(* Logix 5000 project; controller reports 1756-L63 rev 20.11; software revision 20.04; part 4 of 52 *)

        [307].log_data[0].time := 900.0, [307].log_data[0].valid := 1, [307].log_data[1].valid := 1, [307].log_data[2].valid := 1, [307].log_data[3].valid := 1, [307].log_data[4].valid := 1, [307].log_data[5].valid := 1, [307].log_data[6].valid := 1, [307].log_data[7].valid := 1, [307].log_data[8].valid := 1, [307].log_data[9].valid := 1, [307].log_data[10].valid := 1, [307].log_data[11].valid := 1, [307].log_data[12].valid := 1, [307].log_data[13].valid := 1, [307].log_data[14].valid := 1, [307].log_data[15].valid := 1, [307].log_data[16].valid := 1, [307].log_data[17].valid := 1, [307].log_data[18].valid := 1, [307].log_data[19].valid := 1, [307].time.Year := 2023, [307].time.Month := 1, [307].time.Day := 19, [307].time.Hour := 5, [307].time.Minute := 14, [307].time.Second := 59, [308].log_data[0].min := 1.0, [308].log_data[0].max := 1.0, [308].log_data[0].total := 900.0, [308].log_data[0].time := 900.0, [308].log_data[0].minminute := 15, [308].log_data[0].maxminute := 15, [308].log_data[0].valid := 1, [308].log_data[1].valid := 1, [308].log_data[2].valid := 1, [308].log_data[3].valid := 1, [308].log_data[4].valid := 1, [308].log_data[5].valid := 1, [308].log_data[6].valid := 1, [308].log_data[7].valid := 1, [308].log_data[8].valid := 1, [308].log_data[9].valid := 1, [308].log_data[10].valid := 1, [308].log_data[11].valid := 1, [308].log_data[12].valid := 1, [308].log_data[13].valid := 1, [308].log_data[14].valid := 1, [308].log_data[15].valid := 1, [308].log_data[16].valid := 1, [308].log_data[17].valid := 1, [308].log_data[18].valid := 1, [308].log_data[19].valid := 1, [308].time.Year := 2023, [308].time.Month := 1, [308].time.Day := 19, [308].time.Hour := 5, [308].time.Minute := 29, [308].time.Second := 59, [309].log_data[0].min := 1.0,
        [309].log_data[0].max := 1.0, [309].log_data[0].total := 900.0, [309].log_data[0].time := 900.0, [309].log_data[0].minminute := 30, [309].log_data[0].maxminute := 30, [309].log_data[0].valid := 1, [309].log_data[1].valid := 1, [309].log_data[2].valid := 1, [309].log_data[3].valid := 1, [309].log_data[4].valid := 1, [309].log_data[5].valid := 1, [309].log_data[6].valid := 1, [309].log_data[7].valid := 1, [309].log_data[8].valid := 1, [309].log_data[9].valid := 1, [309].log_data[10].valid := 1, [309].log_data[11].valid := 1, [309].log_data[12].valid := 1, [309].log_data[13].valid := 1, [309].log_data[14].valid := 1, [309].log_data[15].valid := 1, [309].log_data[16].valid := 1, [309].log_data[17].valid := 1, [309].log_data[18].valid := 1, [309].log_data[19].valid := 1, [309].time.Year := 2023, [309].time.Month := 1, [309].time.Day := 19, [309].time.Hour := 5, [309].time.Minute := 44, [309].time.Second := 59, [310].log_data[0].min := 1.0, [310].log_data[0].max := 1.0, [310].log_data[0].total := 900.0, [310].log_data[0].time := 900.0, [310].log_data[0].minminute := 45, [310].log_data[0].maxminute := 45, [310].log_data[0].valid := 1, [310].log_data[1].valid := 1, [310].log_data[2].valid := 1, [310].log_data[3].valid := 1, [310].log_data[4].valid := 1, [310].log_data[5].valid := 1, [310].log_data[6].valid := 1, [310].log_data[7].valid := 1, [310].log_data[8].valid := 1, [310].log_data[9].valid := 1, [310].log_data[10].valid := 1, [310].log_data[11].valid := 1, [310].log_data[12].valid := 1, [310].log_data[13].valid := 1, [310].log_data[14].valid := 1, [310].log_data[15].valid := 1, [310].log_data[16].valid := 1, [310].log_data[17].valid := 1, [310].log_data[18].valid := 1, [310].log_data[19].valid := 1, [310].time.Year := 2023, [310].time.Month := 1, [310].time.Day := 19,
        [310].time.Hour := 5, [310].time.Minute := 59, [310].time.Second := 59, [311].log_data[0].min := 1.0, [311].log_data[0].max := 1.0, [311].log_data[0].total := 900.0, [311].log_data[0].time := 900.0, [311].log_data[0].valid := 1, [311].log_data[1].valid := 1, [311].log_data[2].valid := 1, [311].log_data[3].valid := 1, [311].log_data[4].valid := 1, [311].log_data[5].valid := 1, [311].log_data[6].valid := 1, [311].log_data[7].valid := 1, [311].log_data[8].valid := 1, [311].log_data[9].valid := 1, [311].log_data[10].valid := 1, [311].log_data[11].valid := 1, [311].log_data[12].valid := 1, [311].log_data[13].valid := 1, [311].log_data[14].valid := 1, [311].log_data[15].valid := 1, [311].log_data[16].valid := 1, [311].log_data[17].valid := 1, [311].log_data[18].valid := 1, [311].log_data[19].valid := 1, [311].time.Year := 2023, [311].time.Month := 1, [311].time.Day := 19, [311].time.Hour := 6, [311].time.Minute := 14, [311].time.Second := 59, [312].log_data[0].min := 1.0, [312].log_data[0].max := 1.0, [312].log_data[0].total := 900.0, [312].log_data[0].time := 900.0, [312].log_data[0].minminute := 15, [312].log_data[0].maxminute := 15, [312].log_data[0].valid := 1, [312].log_data[1].valid := 1, [312].log_data[2].valid := 1, [312].log_data[3].valid := 1, [312].log_data[4].valid := 1, [312].log_data[5].valid := 1, [312].log_data[6].valid := 1, [312].log_data[7].valid := 1, [312].log_data[8].valid := 1, [312].log_data[9].valid := 1, [312].log_data[10].valid := 1, [312].log_data[11].valid := 1, [312].log_data[12].valid := 1, [312].log_data[13].valid := 1, [312].log_data[14].valid := 1, [312].log_data[15].valid := 1, [312].log_data[16].valid := 1, [312].log_data[17].valid := 1, [312].log_data[18].valid := 1, [312].log_data[19].valid := 1, [312].time.Year := 2023,
        [312].time.Month := 1, [312].time.Day := 19, [312].time.Hour := 6, [312].time.Minute := 29, [312].time.Second := 59, [313].log_data[0].min := 1.0, [313].log_data[0].max := 1.0, [313].log_data[0].total := 900.0, [313].log_data[0].time := 900.0, [313].log_data[0].minminute := 30, [313].log_data[0].maxminute := 30, [313].log_data[0].valid := 1, [313].log_data[1].valid := 1, [313].log_data[2].valid := 1, [313].log_data[3].valid := 1, [313].log_data[4].valid := 1, [313].log_data[5].valid := 1, [313].log_data[6].valid := 1, [313].log_data[7].valid := 1, [313].log_data[8].valid := 1, [313].log_data[9].valid := 1, [313].log_data[10].valid := 1, [313].log_data[11].valid := 1, [313].log_data[12].valid := 1, [313].log_data[13].valid := 1, [313].log_data[14].valid := 1, [313].log_data[15].valid := 1, [313].log_data[16].valid := 1, [313].log_data[17].valid := 1, [313].log_data[18].valid := 1, [313].log_data[19].valid := 1, [313].time.Year := 2023, [313].time.Month := 1, [313].time.Day := 19, [313].time.Hour := 6, [313].time.Minute := 44, [313].time.Second := 59, [314].log_data[0].min := 1.0, [314].log_data[0].max := 1.0, [314].log_data[0].total := 900.0, [314].log_data[0].time := 900.0, [314].log_data[0].minminute := 45, [314].log_data[0].maxminute := 45, [314].log_data[0].valid := 1, [314].log_data[1].valid := 1, [314].log_data[2].valid := 1, [314].log_data[3].valid := 1, [314].log_data[4].valid := 1, [314].log_data[5].valid := 1, [314].log_data[6].valid := 1, [314].log_data[7].valid := 1, [314].log_data[8].valid := 1, [314].log_data[9].valid := 1, [314].log_data[10].valid := 1, [314].log_data[11].valid := 1, [314].log_data[12].valid := 1, [314].log_data[13].valid := 1, [314].log_data[14].valid := 1, [314].log_data[15].valid := 1, [314].log_data[16].valid := 1,
        [314].log_data[17].valid := 1, [314].log_data[18].valid := 1, [314].log_data[19].valid := 1, [314].time.Year := 2023, [314].time.Month := 1, [314].time.Day := 19, [314].time.Hour := 6, [314].time.Minute := 59, [314].time.Second := 59, [315].log_data[0].min := 1.0, [315].log_data[0].max := 1.0, [315].log_data[0].total := 900.0, [315].log_data[0].time := 900.0, [315].log_data[0].valid := 1, [315].log_data[1].valid := 1, [315].log_data[2].valid := 1, [315].log_data[3].valid := 1, [315].log_data[4].valid := 1, [315].log_data[5].valid := 1, [315].log_data[6].valid := 1, [315].log_data[7].valid := 1, [315].log_data[8].valid := 1, [315].log_data[9].valid := 1, [315].log_data[10].valid := 1, [315].log_data[11].valid := 1, [315].log_data[12].valid := 1, [315].log_data[13].valid := 1, [315].log_data[14].valid := 1, [315].log_data[15].valid := 1, [315].log_data[16].valid := 1, [315].log_data[17].valid := 1, [315].log_data[18].valid := 1, [315].log_data[19].valid := 1, [315].time.Year := 2023, [315].time.Month := 1, [315].time.Day := 19, [315].time.Hour := 7, [315].time.Minute := 14, [315].time.Second := 59, [316].log_data[0].min := 1.0, [316].log_data[0].max := 1.0, [316].log_data[0].total := 900.0, [316].log_data[0].time := 900.0, [316].log_data[0].minminute := 15, [316].log_data[0].maxminute := 15, [316].log_data[0].valid := 1, [316].log_data[1].valid := 1, [316].log_data[2].valid := 1, [316].log_data[3].valid := 1, [316].log_data[4].valid := 1, [316].log_data[5].valid := 1, [316].log_data[6].valid := 1, [316].log_data[7].valid := 1, [316].log_data[8].valid := 1, [316].log_data[9].valid := 1, [316].log_data[10].valid := 1, [316].log_data[11].valid := 1, [316].log_data[12].valid := 1, [316].log_data[13].valid := 1, [316].log_data[14].valid := 1,
        [316].log_data[15].valid := 1, [316].log_data[16].valid := 1, [316].log_data[17].valid := 1, [316].log_data[18].valid := 1, [316].log_data[19].valid := 1, [316].time.Year := 2023, [316].time.Month := 1, [316].time.Day := 19, [316].time.Hour := 7, [316].time.Minute := 29, [316].time.Second := 59, [317].log_data[0].min := 1.0, [317].log_data[0].max := 1.0, [317].log_data[0].total := 900.0, [317].log_data[0].time := 900.0, [317].log_data[0].minminute := 30, [317].log_data[0].maxminute := 30, [317].log_data[0].valid := 1, [317].log_data[1].valid := 1, [317].log_data[2].valid := 1, [317].log_data[3].valid := 1, [317].log_data[4].valid := 1, [317].log_data[5].valid := 1, [317].log_data[6].valid := 1, [317].log_data[7].valid := 1, [317].log_data[8].valid := 1, [317].log_data[9].valid := 1, [317].log_data[10].valid := 1, [317].log_data[11].valid := 1, [317].log_data[12].valid := 1, [317].log_data[13].valid := 1, [317].log_data[14].valid := 1, [317].log_data[15].valid := 1, [317].log_data[16].valid := 1, [317].log_data[17].valid := 1, [317].log_data[18].valid := 1, [317].log_data[19].valid := 1, [317].time.Year := 2023, [317].time.Month := 1, [317].time.Day := 19, [317].time.Hour := 7, [317].time.Minute := 44, [317].time.Second := 59, [318].log_data[0].min := 1.0, [318].log_data[0].max := 1.0, [318].log_data[0].total := 900.0, [318].log_data[0].time := 900.0, [318].log_data[0].minminute := 45, [318].log_data[0].maxminute := 45, [318].log_data[0].valid := 1, [318].log_data[1].valid := 1, [318].log_data[2].valid := 1, [318].log_data[3].valid := 1, [318].log_data[4].valid := 1, [318].log_data[5].valid := 1, [318].log_data[6].valid := 1, [318].log_data[7].valid := 1, [318].log_data[8].valid := 1, [318].log_data[9].valid := 1, [318].log_data[10].valid := 1,
        [318].log_data[11].valid := 1, [318].log_data[12].valid := 1, [318].log_data[13].valid := 1, [318].log_data[14].valid := 1, [318].log_data[15].valid := 1, [318].log_data[16].valid := 1, [318].log_data[17].valid := 1, [318].log_data[18].valid := 1, [318].log_data[19].valid := 1, [318].time.Year := 2023, [318].time.Month := 1, [318].time.Day := 19, [318].time.Hour := 7, [318].time.Minute := 59, [318].time.Second := 59, [319].log_data[0].min := 1.0, [319].log_data[0].max := 1.0, [319].log_data[0].total := 899.5, [319].log_data[0].time := 899.5, [319].log_data[0].valid := 1, [319].log_data[1].valid := 1, [319].log_data[2].valid := 1, [319].log_data[3].valid := 1, [319].log_data[4].valid := 1, [319].log_data[5].valid := 1, [319].log_data[6].valid := 1, [319].log_data[7].valid := 1, [319].log_data[8].valid := 1, [319].log_data[9].valid := 1, [319].log_data[10].valid := 1, [319].log_data[11].valid := 1, [319].log_data[12].valid := 1, [319].log_data[13].valid := 1, [319].log_data[14].valid := 1, [319].log_data[15].valid := 1, [319].log_data[16].valid := 1, [319].log_data[17].valid := 1, [319].log_data[18].valid := 1, [319].log_data[19].valid := 1, [319].time.Year := 2023, [319].time.Month := 1, [319].time.Day := 19, [319].time.Hour := 8, [319].time.Minute := 14, [319].time.Second := 59, [320].log_data[0].min := 1.0, [320].log_data[0].max := 1.0, [320].log_data[0].total := 900.0, [320].log_data[0].time := 900.0, [320].log_data[0].minminute := 15, [320].log_data[0].maxminute := 15, [320].log_data[0].valid := 1, [320].log_data[1].valid := 1, [320].log_data[2].valid := 1, [320].log_data[3].valid := 1, [320].log_data[4].valid := 1, [320].log_data[5].valid := 1, [320].log_data[6].valid := 1, [320].log_data[7].valid := 1, [320].log_data[8].valid := 1,
        [320].log_data[9].valid := 1, [320].log_data[10].valid := 1, [320].log_data[11].valid := 1, [320].log_data[12].valid := 1, [320].log_data[13].valid := 1, [320].log_data[14].valid := 1, [320].log_data[15].valid := 1, [320].log_data[16].valid := 1, [320].log_data[17].valid := 1, [320].log_data[18].valid := 1, [320].log_data[19].valid := 1, [320].time.Year := 2023, [320].time.Month := 1, [320].time.Day := 19, [320].time.Hour := 8, [320].time.Minute := 29, [320].time.Second := 59, [321].log_data[0].min := 1.0, [321].log_data[0].max := 1.0, [321].log_data[0].total := 900.0, [321].log_data[0].time := 900.0, [321].log_data[0].minminute := 30, [321].log_data[0].maxminute := 30, [321].log_data[0].valid := 1, [321].log_data[1].valid := 1, [321].log_data[2].valid := 1, [321].log_data[3].valid := 1, [321].log_data[4].valid := 1, [321].log_data[5].valid := 1, [321].log_data[6].valid := 1, [321].log_data[7].valid := 1, [321].log_data[8].valid := 1, [321].log_data[9].valid := 1, [321].log_data[10].valid := 1, [321].log_data[11].valid := 1, [321].log_data[12].valid := 1, [321].log_data[13].valid := 1, [321].log_data[14].valid := 1, [321].log_data[15].valid := 1, [321].log_data[16].valid := 1, [321].log_data[17].valid := 1, [321].log_data[18].valid := 1, [321].log_data[19].valid := 1, [321].time.Year := 2023, [321].time.Month := 1, [321].time.Day := 19, [321].time.Hour := 8, [321].time.Minute := 44, [321].time.Second := 59, [322].log_data[0].min := 1.0, [322].log_data[0].max := 1.0, [322].log_data[0].total := 900.0, [322].log_data[0].time := 900.0, [322].log_data[0].minminute := 45, [322].log_data[0].maxminute := 45, [322].log_data[0].valid := 1, [322].log_data[1].valid := 1, [322].log_data[2].valid := 1, [322].log_data[3].valid := 1, [322].log_data[4].valid := 1,
        [322].log_data[5].valid := 1, [322].log_data[6].valid := 1, [322].log_data[7].valid := 1, [322].log_data[8].valid := 1, [322].log_data[9].valid := 1, [322].log_data[10].valid := 1, [322].log_data[11].valid := 1, [322].log_data[12].valid := 1, [322].log_data[13].valid := 1, [322].log_data[14].valid := 1, [322].log_data[15].valid := 1, [322].log_data[16].valid := 1, [322].log_data[17].valid := 1, [322].log_data[18].valid := 1, [322].log_data[19].valid := 1, [322].time.Year := 2023, [322].time.Month := 1, [322].time.Day := 19, [322].time.Hour := 8, [322].time.Minute := 59, [322].time.Second := 59, [323].log_data[0].min := 1.0, [323].log_data[0].max := 1.0, [323].log_data[0].total := 900.0, [323].log_data[0].time := 900.0, [323].log_data[0].valid := 1, [323].log_data[1].valid := 1, [323].log_data[2].valid := 1, [323].log_data[3].valid := 1, [323].log_data[4].valid := 1, [323].log_data[5].valid := 1, [323].log_data[6].valid := 1, [323].log_data[7].valid := 1, [323].log_data[8].valid := 1, [323].log_data[9].valid := 1, [323].log_data[10].valid := 1, [323].log_data[11].valid := 1, [323].log_data[12].valid := 1, [323].log_data[13].valid := 1, [323].log_data[14].valid := 1, [323].log_data[15].valid := 1, [323].log_data[16].valid := 1, [323].log_data[17].valid := 1, [323].log_data[18].valid := 1, [323].log_data[19].valid := 1, [323].time.Year := 2023, [323].time.Month := 1, [323].time.Day := 19, [323].time.Hour := 9, [323].time.Minute := 14, [323].time.Second := 59, [324].log_data[0].min := 1.0, [324].log_data[0].max := 1.0, [324].log_data[0].total := 900.0, [324].log_data[0].time := 900.0, [324].log_data[0].minminute := 15, [324].log_data[0].maxminute := 15, [324].log_data[0].valid := 1, [324].log_data[1].valid := 1, [324].log_data[2].valid := 1,
        [324].log_data[3].valid := 1, [324].log_data[4].valid := 1, [324].log_data[5].valid := 1, [324].log_data[6].valid := 1, [324].log_data[7].valid := 1, [324].log_data[8].valid := 1, [324].log_data[9].valid := 1, [324].log_data[10].valid := 1, [324].log_data[11].valid := 1, [324].log_data[12].valid := 1, [324].log_data[13].valid := 1, [324].log_data[14].valid := 1, [324].log_data[15].valid := 1, [324].log_data[16].valid := 1, [324].log_data[17].valid := 1, [324].log_data[18].valid := 1, [324].log_data[19].valid := 1, [324].time.Year := 2023, [324].time.Month := 1, [324].time.Day := 19, [324].time.Hour := 9, [324].time.Minute := 29, [324].time.Second := 59, [325].log_data[0].min := 1.0, [325].log_data[0].max := 1.0, [325].log_data[0].total := 900.0, [325].log_data[0].time := 900.0, [325].log_data[0].minminute := 30, [325].log_data[0].maxminute := 30, [325].log_data[0].valid := 1, [325].log_data[1].valid := 1, [325].log_data[2].valid := 1, [325].log_data[3].valid := 1, [325].log_data[4].valid := 1, [325].log_data[5].valid := 1, [325].log_data[6].valid := 1, [325].log_data[7].valid := 1, [325].log_data[8].valid := 1, [325].log_data[9].valid := 1, [325].log_data[10].valid := 1, [325].log_data[11].valid := 1, [325].log_data[12].valid := 1, [325].log_data[13].valid := 1, [325].log_data[14].valid := 1, [325].log_data[15].valid := 1, [325].log_data[16].valid := 1, [325].log_data[17].valid := 1, [325].log_data[18].valid := 1, [325].log_data[19].valid := 1, [325].time.Year := 2023, [325].time.Month := 1, [325].time.Day := 19, [325].time.Hour := 9, [325].time.Minute := 44, [325].time.Second := 59, [326].log_data[0].min := 1.0, [326].log_data[0].max := 1.0, [326].log_data[0].total := 900.0, [326].log_data[0].time := 900.0, [326].log_data[0].minminute := 45,
        [326].log_data[0].maxminute := 45, [326].log_data[0].valid := 1, [326].log_data[1].valid := 1, [326].log_data[2].valid := 1, [326].log_data[3].valid := 1, [326].log_data[4].valid := 1, [326].log_data[5].valid := 1, [326].log_data[6].valid := 1, [326].log_data[7].valid := 1, [326].log_data[8].valid := 1, [326].log_data[9].valid := 1, [326].log_data[10].valid := 1, [326].log_data[11].valid := 1, [326].log_data[12].valid := 1, [326].log_data[13].valid := 1, [326].log_data[14].valid := 1, [326].log_data[15].valid := 1, [326].log_data[16].valid := 1, [326].log_data[17].valid := 1, [326].log_data[18].valid := 1, [326].log_data[19].valid := 1, [326].time.Year := 2023, [326].time.Month := 1, [326].time.Day := 19, [326].time.Hour := 9, [326].time.Minute := 59, [326].time.Second := 59, [327].log_data[0].min := 1.0, [327].log_data[0].max := 1.0, [327].log_data[0].total := 900.0, [327].log_data[0].time := 900.0, [327].log_data[0].valid := 1, [327].log_data[1].valid := 1, [327].log_data[2].valid := 1, [327].log_data[3].valid := 1, [327].log_data[4].valid := 1, [327].log_data[5].valid := 1, [327].log_data[6].valid := 1, [327].log_data[7].valid := 1, [327].log_data[8].valid := 1, [327].log_data[9].valid := 1, [327].log_data[10].valid := 1, [327].log_data[11].valid := 1, [327].log_data[12].valid := 1, [327].log_data[13].valid := 1, [327].log_data[14].valid := 1, [327].log_data[15].valid := 1, [327].log_data[16].valid := 1, [327].log_data[17].valid := 1, [327].log_data[18].valid := 1, [327].log_data[19].valid := 1, [327].time.Year := 2023, [327].time.Month := 1, [327].time.Day := 19, [327].time.Hour := 10, [327].time.Minute := 14, [327].time.Second := 59, [328].log_data[0].min := 1.0, [328].log_data[0].max := 1.0, [328].log_data[0].total := 900.0,
        [328].log_data[0].time := 900.0, [328].log_data[0].minminute := 15, [328].log_data[0].maxminute := 15, [328].log_data[0].valid := 1, [328].log_data[1].valid := 1, [328].log_data[2].valid := 1, [328].log_data[3].valid := 1, [328].log_data[4].valid := 1, [328].log_data[5].valid := 1, [328].log_data[6].valid := 1, [328].log_data[7].valid := 1, [328].log_data[8].valid := 1, [328].log_data[9].valid := 1, [328].log_data[10].valid := 1, [328].log_data[11].valid := 1, [328].log_data[12].valid := 1, [328].log_data[13].valid := 1, [328].log_data[14].valid := 1, [328].log_data[15].valid := 1, [328].log_data[16].valid := 1, [328].log_data[17].valid := 1, [328].log_data[18].valid := 1, [328].log_data[19].valid := 1, [328].time.Year := 2023, [328].time.Month := 1, [328].time.Day := 19, [328].time.Hour := 10, [328].time.Minute := 29, [328].time.Second := 59, [329].log_data[0].min := 1.0, [329].log_data[0].max := 1.0, [329].log_data[0].total := 900.0, [329].log_data[0].time := 900.0, [329].log_data[0].minminute := 30, [329].log_data[0].maxminute := 30, [329].log_data[0].valid := 1, [329].log_data[1].valid := 1, [329].log_data[2].valid := 1, [329].log_data[3].valid := 1, [329].log_data[4].valid := 1, [329].log_data[5].valid := 1, [329].log_data[6].valid := 1, [329].log_data[7].valid := 1, [329].log_data[8].valid := 1, [329].log_data[9].valid := 1, [329].log_data[10].valid := 1, [329].log_data[11].valid := 1, [329].log_data[12].valid := 1, [329].log_data[13].valid := 1, [329].log_data[14].valid := 1, [329].log_data[15].valid := 1, [329].log_data[16].valid := 1, [329].log_data[17].valid := 1, [329].log_data[18].valid := 1, [329].log_data[19].valid := 1, [329].time.Year := 2023, [329].time.Month := 1, [329].time.Day := 19, [329].time.Hour := 10, [329].time.Minute := 44,
        [329].time.Second := 59, [330].log_data[0].min := 1.0, [330].log_data[0].max := 1.0, [330].log_data[0].total := 900.0, [330].log_data[0].time := 900.0, [330].log_data[0].minminute := 45, [330].log_data[0].maxminute := 45, [330].log_data[0].valid := 1, [330].log_data[1].valid := 1, [330].log_data[2].valid := 1, [330].log_data[3].valid := 1, [330].log_data[4].valid := 1, [330].log_data[5].valid := 1, [330].log_data[6].valid := 1, [330].log_data[7].valid := 1, [330].log_data[8].valid := 1, [330].log_data[9].valid := 1, [330].log_data[10].valid := 1, [330].log_data[11].valid := 1, [330].log_data[12].valid := 1, [330].log_data[13].valid := 1, [330].log_data[14].valid := 1, [330].log_data[15].valid := 1, [330].log_data[16].valid := 1, [330].log_data[17].valid := 1, [330].log_data[18].valid := 1, [330].log_data[19].valid := 1, [330].time.Year := 2023, [330].time.Month := 1, [330].time.Day := 19, [330].time.Hour := 10, [330].time.Minute := 59, [330].time.Second := 59, [331].log_data[0].min := 1.0, [331].log_data[0].max := 1.0, [331].log_data[0].total := 900.0, [331].log_data[0].time := 900.0, [331].log_data[0].valid := 1, [331].log_data[1].valid := 1, [331].log_data[2].valid := 1, [331].log_data[3].valid := 1, [331].log_data[4].valid := 1, [331].log_data[5].valid := 1, [331].log_data[6].valid := 1, [331].log_data[7].valid := 1, [331].log_data[8].valid := 1, [331].log_data[9].valid := 1, [331].log_data[10].valid := 1, [331].log_data[11].valid := 1, [331].log_data[12].valid := 1, [331].log_data[13].valid := 1, [331].log_data[14].valid := 1, [331].log_data[15].valid := 1, [331].log_data[16].valid := 1, [331].log_data[17].valid := 1, [331].log_data[18].valid := 1, [331].log_data[19].valid := 1, [331].time.Year := 2023, [331].time.Month := 1, [331].time.Day := 19,
        [331].time.Hour := 11, [331].time.Minute := 14, [331].time.Second := 59, [332].log_data[0].min := 1.0, [332].log_data[0].max := 1.0, [332].log_data[0].total := 900.0, [332].log_data[0].time := 900.0, [332].log_data[0].minminute := 15, [332].log_data[0].maxminute := 15, [332].log_data[0].valid := 1, [332].log_data[1].valid := 1, [332].log_data[2].valid := 1, [332].log_data[3].valid := 1, [332].log_data[4].valid := 1, [332].log_data[5].valid := 1, [332].log_data[6].valid := 1, [332].log_data[7].valid := 1, [332].log_data[8].valid := 1, [332].log_data[9].valid := 1, [332].log_data[10].valid := 1, [332].log_data[11].valid := 1, [332].log_data[12].valid := 1, [332].log_data[13].valid := 1, [332].log_data[14].valid := 1, [332].log_data[15].valid := 1, [332].log_data[16].valid := 1, [332].log_data[17].valid := 1, [332].log_data[18].valid := 1, [332].log_data[19].valid := 1, [332].time.Year := 2023, [332].time.Month := 1, [332].time.Day := 19, [332].time.Hour := 11, [332].time.Minute := 29, [332].time.Second := 59, [333].log_data[0].min := 1.0, [333].log_data[0].max := 1.0, [333].log_data[0].total := 900.0, [333].log_data[0].time := 900.0, [333].log_data[0].minminute := 30, [333].log_data[0].maxminute := 30, [333].log_data[0].valid := 1, [333].log_data[1].valid := 1, [333].log_data[2].valid := 1, [333].log_data[3].valid := 1, [333].log_data[4].valid := 1, [333].log_data[5].valid := 1, [333].log_data[6].valid := 1, [333].log_data[7].valid := 1, [333].log_data[8].valid := 1, [333].log_data[9].valid := 1, [333].log_data[10].valid := 1, [333].log_data[11].valid := 1, [333].log_data[12].valid := 1, [333].log_data[13].valid := 1, [333].log_data[14].valid := 1, [333].log_data[15].valid := 1, [333].log_data[16].valid := 1, [333].log_data[17].valid := 1, [333].log_data[18].valid := 1,
        [333].log_data[19].valid := 1, [333].time.Year := 2023, [333].time.Month := 1, [333].time.Day := 19, [333].time.Hour := 11, [333].time.Minute := 44, [333].time.Second := 59, [334].log_data[0].min := 1.0, [334].log_data[0].max := 1.0, [334].log_data[0].total := 900.0, [334].log_data[0].time := 900.0, [334].log_data[0].minminute := 45, [334].log_data[0].maxminute := 45, [334].log_data[0].valid := 1, [334].log_data[1].valid := 1, [334].log_data[2].valid := 1, [334].log_data[3].valid := 1, [334].log_data[4].valid := 1, [334].log_data[5].valid := 1, [334].log_data[6].valid := 1, [334].log_data[7].valid := 1, [334].log_data[8].valid := 1, [334].log_data[9].valid := 1, [334].log_data[10].valid := 1, [334].log_data[11].valid := 1, [334].log_data[12].valid := 1, [334].log_data[13].valid := 1, [334].log_data[14].valid := 1, [334].log_data[15].valid := 1, [334].log_data[16].valid := 1, [334].log_data[17].valid := 1, [334].log_data[18].valid := 1, [334].log_data[19].valid := 1, [334].time.Year := 2023, [334].time.Month := 1, [334].time.Day := 19, [334].time.Hour := 11, [334].time.Minute := 59, [334].time.Second := 59, [335].log_data[0].min := 1.0, [335].log_data[0].max := 1.0, [335].log_data[0].total := 900.0, [335].log_data[0].time := 900.0, [335].log_data[0].valid := 1, [335].log_data[1].valid := 1, [335].log_data[2].valid := 1, [335].log_data[3].valid := 1, [335].log_data[4].valid := 1, [335].log_data[5].valid := 1, [335].log_data[6].valid := 1, [335].log_data[7].valid := 1, [335].log_data[8].valid := 1, [335].log_data[9].valid := 1, [335].log_data[10].valid := 1, [335].log_data[11].valid := 1, [335].log_data[12].valid := 1, [335].log_data[13].valid := 1, [335].log_data[14].valid := 1, [335].log_data[15].valid := 1, [335].log_data[16].valid := 1,
        [335].log_data[17].valid := 1, [335].log_data[18].valid := 1, [335].log_data[19].valid := 1, [335].time.Year := 2023, [335].time.Month := 1, [335].time.Day := 19, [335].time.Hour := 12, [335].time.Minute := 14, [335].time.Second := 59, [336].log_data[0].min := 1.0, [336].log_data[0].max := 1.0, [336].log_data[0].total := 900.0, [336].log_data[0].time := 900.0, [336].log_data[0].minminute := 15, [336].log_data[0].maxminute := 15, [336].log_data[0].valid := 1, [336].log_data[1].valid := 1, [336].log_data[2].valid := 1, [336].log_data[3].valid := 1, [336].log_data[4].valid := 1, [336].log_data[5].valid := 1, [336].log_data[6].valid := 1, [336].log_data[7].valid := 1, [336].log_data[8].valid := 1, [336].log_data[9].valid := 1, [336].log_data[10].valid := 1, [336].log_data[11].valid := 1, [336].log_data[12].valid := 1, [336].log_data[13].valid := 1, [336].log_data[14].valid := 1, [336].log_data[15].valid := 1, [336].log_data[16].valid := 1, [336].log_data[17].valid := 1, [336].log_data[18].valid := 1, [336].log_data[19].valid := 1, [336].time.Year := 2023, [336].time.Month := 1, [336].time.Day := 19, [336].time.Hour := 12, [336].time.Minute := 29, [336].time.Second := 59, [337].log_data[0].min := 1.0, [337].log_data[0].max := 1.0, [337].log_data[0].total := 900.0, [337].log_data[0].time := 900.0, [337].log_data[0].minminute := 30, [337].log_data[0].maxminute := 30, [337].log_data[0].valid := 1, [337].log_data[1].valid := 1, [337].log_data[2].valid := 1, [337].log_data[3].valid := 1, [337].log_data[4].valid := 1, [337].log_data[5].valid := 1, [337].log_data[6].valid := 1, [337].log_data[7].valid := 1, [337].log_data[8].valid := 1, [337].log_data[9].valid := 1, [337].log_data[10].valid := 1, [337].log_data[11].valid := 1, [337].log_data[12].valid := 1,
        [337].log_data[13].valid := 1, [337].log_data[14].valid := 1, [337].log_data[15].valid := 1, [337].log_data[16].valid := 1, [337].log_data[17].valid := 1, [337].log_data[18].valid := 1, [337].log_data[19].valid := 1, [337].time.Year := 2023, [337].time.Month := 1, [337].time.Day := 19, [337].time.Hour := 12, [337].time.Minute := 44, [337].time.Second := 59, [338].log_data[0].min := 1.0, [338].log_data[0].max := 1.0, [338].log_data[0].total := 900.0, [338].log_data[0].time := 900.0, [338].log_data[0].minminute := 45, [338].log_data[0].maxminute := 45, [338].log_data[0].valid := 1, [338].log_data[1].valid := 1, [338].log_data[2].valid := 1, [338].log_data[3].valid := 1, [338].log_data[4].valid := 1, [338].log_data[5].valid := 1, [338].log_data[6].valid := 1, [338].log_data[7].valid := 1, [338].log_data[8].valid := 1, [338].log_data[9].valid := 1, [338].log_data[10].valid := 1, [338].log_data[11].valid := 1, [338].log_data[12].valid := 1, [338].log_data[13].valid := 1, [338].log_data[14].valid := 1, [338].log_data[15].valid := 1, [338].log_data[16].valid := 1, [338].log_data[17].valid := 1, [338].log_data[18].valid := 1, [338].log_data[19].valid := 1, [338].time.Year := 2023, [338].time.Month := 1, [338].time.Day := 19, [338].time.Hour := 12, [338].time.Minute := 59, [338].time.Second := 59, [339].log_data[0].min := 1.0, [339].log_data[0].max := 1.0, [339].log_data[0].total := 900.0, [339].log_data[0].time := 900.0, [339].log_data[0].valid := 1, [339].log_data[1].valid := 1, [339].log_data[2].valid := 1, [339].log_data[3].valid := 1, [339].log_data[4].valid := 1, [339].log_data[5].valid := 1, [339].log_data[6].valid := 1, [339].log_data[7].valid := 1, [339].log_data[8].valid := 1, [339].log_data[9].valid := 1, [339].log_data[10].valid := 1,
        [339].log_data[11].valid := 1, [339].log_data[12].valid := 1, [339].log_data[13].valid := 1, [339].log_data[14].valid := 1, [339].log_data[15].valid := 1, [339].log_data[16].valid := 1, [339].log_data[17].valid := 1, [339].log_data[18].valid := 1, [339].log_data[19].valid := 1, [339].time.Year := 2023, [339].time.Month := 1, [339].time.Day := 19, [339].time.Hour := 13, [339].time.Minute := 14, [339].time.Second := 59, [340].log_data[0].min := 1.0, [340].log_data[0].max := 1.0, [340].log_data[0].total := 900.0, [340].log_data[0].time := 900.0, [340].log_data[0].minminute := 15, [340].log_data[0].maxminute := 15, [340].log_data[0].valid := 1, [340].log_data[1].valid := 1, [340].log_data[2].valid := 1, [340].log_data[3].valid := 1, [340].log_data[4].valid := 1, [340].log_data[5].valid := 1, [340].log_data[6].valid := 1, [340].log_data[7].valid := 1, [340].log_data[8].valid := 1, [340].log_data[9].valid := 1, [340].log_data[10].valid := 1, [340].log_data[11].valid := 1, [340].log_data[12].valid := 1, [340].log_data[13].valid := 1, [340].log_data[14].valid := 1, [340].log_data[15].valid := 1, [340].log_data[16].valid := 1, [340].log_data[17].valid := 1, [340].log_data[18].valid := 1, [340].log_data[19].valid := 1, [340].time.Year := 2023, [340].time.Month := 1, [340].time.Day := 19, [340].time.Hour := 13, [340].time.Minute := 29, [340].time.Second := 59, [341].log_data[0].min := 1.0, [341].log_data[0].max := 1.0, [341].log_data[0].total := 900.0, [341].log_data[0].time := 900.0, [341].log_data[0].minminute := 30, [341].log_data[0].maxminute := 30, [341].log_data[0].valid := 1, [341].log_data[1].valid := 1, [341].log_data[2].valid := 1, [341].log_data[3].valid := 1, [341].log_data[4].valid := 1, [341].log_data[5].valid := 1, [341].log_data[6].valid := 1,
        [341].log_data[7].valid := 1, [341].log_data[8].valid := 1, [341].log_data[9].valid := 1, [341].log_data[10].valid := 1, [341].log_data[11].valid := 1, [341].log_data[12].valid := 1, [341].log_data[13].valid := 1, [341].log_data[14].valid := 1, [341].log_data[15].valid := 1, [341].log_data[16].valid := 1, [341].log_data[17].valid := 1, [341].log_data[18].valid := 1, [341].log_data[19].valid := 1, [341].time.Year := 2023, [341].time.Month := 1, [341].time.Day := 19, [341].time.Hour := 13, [341].time.Minute := 44, [341].time.Second := 59, [342].log_data[0].min := 1.0, [342].log_data[0].max := 1.0, [342].log_data[0].total := 900.0, [342].log_data[0].time := 900.0, [342].log_data[0].minminute := 45, [342].log_data[0].maxminute := 45, [342].log_data[0].valid := 1, [342].log_data[1].valid := 1, [342].log_data[2].valid := 1, [342].log_data[3].valid := 1, [342].log_data[4].valid := 1, [342].log_data[5].valid := 1, [342].log_data[6].valid := 1, [342].log_data[7].valid := 1, [342].log_data[8].valid := 1, [342].log_data[9].valid := 1, [342].log_data[10].valid := 1, [342].log_data[11].valid := 1, [342].log_data[12].valid := 1, [342].log_data[13].valid := 1, [342].log_data[14].valid := 1, [342].log_data[15].valid := 1, [342].log_data[16].valid := 1, [342].log_data[17].valid := 1, [342].log_data[18].valid := 1, [342].log_data[19].valid := 1, [342].time.Year := 2023, [342].time.Month := 1, [342].time.Day := 19, [342].time.Hour := 13, [342].time.Minute := 59, [342].time.Second := 59, [343].log_data[0].min := 1.0, [343].log_data[0].max := 1.0, [343].log_data[0].total := 900.0, [343].log_data[0].time := 900.0, [343].log_data[0].valid := 1, [343].log_data[1].valid := 1, [343].log_data[2].valid := 1, [343].log_data[3].valid := 1, [343].log_data[4].valid := 1,
        [343].log_data[5].valid := 1, [343].log_data[6].valid := 1, [343].log_data[7].valid := 1, [343].log_data[8].valid := 1, [343].log_data[9].valid := 1, [343].log_data[10].valid := 1, [343].log_data[11].valid := 1, [343].log_data[12].valid := 1, [343].log_data[13].valid := 1, [343].log_data[14].valid := 1, [343].log_data[15].valid := 1, [343].log_data[16].valid := 1, [343].log_data[17].valid := 1, [343].log_data[18].valid := 1, [343].log_data[19].valid := 1, [343].time.Year := 2023, [343].time.Month := 1, [343].time.Day := 19, [343].time.Hour := 14, [343].time.Minute := 14, [343].time.Second := 59, [344].log_data[0].min := 1.0, [344].log_data[0].max := 1.0, [344].log_data[0].total := 900.0, [344].log_data[0].time := 900.0, [344].log_data[0].minminute := 15, [344].log_data[0].maxminute := 15, [344].log_data[0].valid := 1, [344].log_data[1].valid := 1, [344].log_data[2].valid := 1, [344].log_data[3].valid := 1, [344].log_data[4].valid := 1, [344].log_data[5].valid := 1, [344].log_data[6].valid := 1, [344].log_data[7].valid := 1, [344].log_data[8].valid := 1, [344].log_data[9].valid := 1, [344].log_data[10].valid := 1, [344].log_data[11].valid := 1, [344].log_data[12].valid := 1, [344].log_data[13].valid := 1, [344].log_data[14].valid := 1, [344].log_data[15].valid := 1, [344].log_data[16].valid := 1, [344].log_data[17].valid := 1, [344].log_data[18].valid := 1, [344].log_data[19].valid := 1, [344].time.Year := 2023, [344].time.Month := 1, [344].time.Day := 19, [344].time.Hour := 14, [344].time.Minute := 29, [344].time.Second := 59, [345].log_data[0].min := 1.0, [345].log_data[0].max := 1.0, [345].log_data[0].total := 900.0, [345].log_data[0].time := 900.0, [345].log_data[0].minminute := 30, [345].log_data[0].maxminute := 30, [345].log_data[0].valid := 1,
        [345].log_data[1].valid := 1, [345].log_data[2].valid := 1, [345].log_data[3].valid := 1, [345].log_data[4].valid := 1, [345].log_data[5].valid := 1, [345].log_data[6].valid := 1, [345].log_data[7].valid := 1, [345].log_data[8].valid := 1, [345].log_data[9].valid := 1, [345].log_data[10].valid := 1, [345].log_data[11].valid := 1, [345].log_data[12].valid := 1, [345].log_data[13].valid := 1, [345].log_data[14].valid := 1, [345].log_data[15].valid := 1, [345].log_data[16].valid := 1, [345].log_data[17].valid := 1, [345].log_data[18].valid := 1, [345].log_data[19].valid := 1, [345].time.Year := 2023, [345].time.Month := 1, [345].time.Day := 19, [345].time.Hour := 14, [345].time.Minute := 44, [345].time.Second := 59, [346].log_data[0].min := 1.0, [346].log_data[0].max := 1.0, [346].log_data[0].total := 900.0, [346].log_data[0].time := 900.0, [346].log_data[0].minminute := 45, [346].log_data[0].maxminute := 45, [346].log_data[0].valid := 1, [346].log_data[1].valid := 1, [346].log_data[2].valid := 1, [346].log_data[3].valid := 1, [346].log_data[4].valid := 1, [346].log_data[5].valid := 1, [346].log_data[6].valid := 1, [346].log_data[7].valid := 1, [346].log_data[8].valid := 1, [346].log_data[9].valid := 1, [346].log_data[10].valid := 1, [346].log_data[11].valid := 1, [346].log_data[12].valid := 1, [346].log_data[13].valid := 1, [346].log_data[14].valid := 1, [346].log_data[15].valid := 1, [346].log_data[16].valid := 1, [346].log_data[17].valid := 1, [346].log_data[18].valid := 1, [346].log_data[19].valid := 1, [346].time.Year := 2023, [346].time.Month := 1, [346].time.Day := 19, [346].time.Hour := 14, [346].time.Minute := 59, [346].time.Second := 59, [347].log_data[0].min := 1.0, [347].log_data[0].max := 1.0, [347].log_data[0].total := 900.0,
        [347].log_data[0].time := 900.0, [347].log_data[0].valid := 1, [347].log_data[1].valid := 1, [347].log_data[2].valid := 1, [347].log_data[3].valid := 1, [347].log_data[4].valid := 1, [347].log_data[5].valid := 1, [347].log_data[6].valid := 1, [347].log_data[7].valid := 1, [347].log_data[8].valid := 1, [347].log_data[9].valid := 1, [347].log_data[10].valid := 1, [347].log_data[11].valid := 1, [347].log_data[12].valid := 1, [347].log_data[13].valid := 1, [347].log_data[14].valid := 1, [347].log_data[15].valid := 1, [347].log_data[16].valid := 1, [347].log_data[17].valid := 1, [347].log_data[18].valid := 1, [347].log_data[19].valid := 1, [347].time.Year := 2023, [347].time.Month := 1, [347].time.Day := 19, [347].time.Hour := 15, [347].time.Minute := 14, [347].time.Second := 59, [348].log_data[0].min := 1.0, [348].log_data[0].max := 1.0, [348].log_data[0].total := 661.251, [348].log_data[0].time := 661.251, [348].log_data[0].minminute := 15, [348].log_data[0].maxminute := 15, [348].log_data[0].valid := 1, [348].log_data[1].valid := 1, [348].log_data[2].valid := 1, [348].log_data[3].valid := 1, [348].log_data[4].valid := 1, [348].log_data[5].valid := 1, [348].log_data[6].valid := 1, [348].log_data[7].valid := 1, [348].log_data[8].valid := 1, [348].log_data[9].valid := 1, [348].log_data[10].valid := 1, [348].log_data[11].valid := 1, [348].log_data[12].valid := 1, [348].log_data[13].valid := 1, [348].log_data[14].valid := 1, [348].log_data[15].valid := 1, [348].log_data[16].valid := 1, [348].log_data[17].valid := 1, [348].log_data[18].valid := 1, [348].log_data[19].valid := 1, [349].log_data[0].min := 1.0, [349].log_data[0].max := 1.0, [349].log_data[0].total := 900.0, [349].log_data[0].time := 900.0, [349].log_data[0].minminute := 30, [349].log_data[0].maxminute := 30, [349].log_data[0].valid := 1,
        [349].log_data[1].valid := 1, [349].log_data[2].valid := 1, [349].log_data[3].valid := 1, [349].log_data[4].valid := 1, [349].log_data[5].valid := 1, [349].log_data[6].valid := 1, [349].log_data[7].valid := 1, [349].log_data[8].valid := 1, [349].log_data[9].valid := 1, [349].log_data[10].valid := 1, [349].log_data[11].valid := 1, [349].log_data[12].valid := 1, [349].log_data[13].valid := 1, [349].log_data[14].valid := 1, [349].log_data[15].valid := 1, [349].log_data[16].valid := 1, [349].log_data[17].valid := 1, [349].log_data[18].valid := 1, [349].log_data[19].valid := 1, [349].time.Year := 2023, [349].time.Month := 1, [349].time.Day := 11, [349].time.Hour := 7, [349].time.Minute := 44, [349].time.Second := 59, [350].log_data[0].min := 1.0, [350].log_data[0].max := 1.0, [350].log_data[0].total := 900.0, [350].log_data[0].time := 900.0, [350].log_data[0].minminute := 45, [350].log_data[0].maxminute := 45, [350].log_data[0].valid := 1, [350].log_data[1].valid := 1, [350].log_data[2].valid := 1, [350].log_data[3].valid := 1, [350].log_data[4].valid := 1, [350].log_data[5].valid := 1, [350].log_data[6].valid := 1, [350].log_data[7].valid := 1, [350].log_data[8].valid := 1, [350].log_data[9].valid := 1, [350].log_data[10].valid := 1, [350].log_data[11].valid := 1, [350].log_data[12].valid := 1, [350].log_data[13].valid := 1, [350].log_data[14].valid := 1, [350].log_data[15].valid := 1, [350].log_data[16].valid := 1, [350].log_data[17].valid := 1, [350].log_data[18].valid := 1, [350].log_data[19].valid := 1, [350].time.Year := 2023, [350].time.Month := 1, [350].time.Day := 11, [350].time.Hour := 7, [350].time.Minute := 59, [350].time.Second := 59, [351].log_data[0].min := 1.0, [351].log_data[0].max := 1.0, [351].log_data[0].total := 900.0,
        [351].log_data[0].time := 900.0, [351].log_data[0].valid := 1, [351].log_data[1].valid := 1, [351].log_data[2].valid := 1, [351].log_data[3].valid := 1, [351].log_data[4].valid := 1, [351].log_data[5].valid := 1, [351].log_data[6].valid := 1, [351].log_data[7].valid := 1, [351].log_data[8].valid := 1, [351].log_data[9].valid := 1, [351].log_data[10].valid := 1, [351].log_data[11].valid := 1, [351].log_data[12].valid := 1, [351].log_data[13].valid := 1, [351].log_data[14].valid := 1, [351].log_data[15].valid := 1, [351].log_data[16].valid := 1, [351].log_data[17].valid := 1, [351].log_data[18].valid := 1, [351].log_data[19].valid := 1, [351].time.Year := 2023, [351].time.Month := 1, [351].time.Day := 11, [351].time.Hour := 8, [351].time.Minute := 14, [351].time.Second := 59, [352].log_data[0].min := 1.0, [352].log_data[0].max := 1.0, [352].log_data[0].total := 900.0, [352].log_data[0].time := 900.0, [352].log_data[0].minminute := 15, [352].log_data[0].maxminute := 15, [352].log_data[0].valid := 1, [352].log_data[1].valid := 1, [352].log_data[2].valid := 1, [352].log_data[3].valid := 1, [352].log_data[4].valid := 1, [352].log_data[5].valid := 1, [352].log_data[6].valid := 1, [352].log_data[7].valid := 1, [352].log_data[8].valid := 1, [352].log_data[9].valid := 1, [352].log_data[10].valid := 1, [352].log_data[11].valid := 1, [352].log_data[12].valid := 1, [352].log_data[13].valid := 1, [352].log_data[14].valid := 1, [352].log_data[15].valid := 1, [352].log_data[16].valid := 1, [352].log_data[17].valid := 1, [352].log_data[18].valid := 1, [352].log_data[19].valid := 1, [352].time.Year := 2023, [352].time.Month := 1, [352].time.Day := 11, [352].time.Hour := 8, [352].time.Minute := 29, [352].time.Second := 59, [353].log_data[0].min := 1.0,
        [353].log_data[0].max := 1.0, [353].log_data[0].total := 900.0, [353].log_data[0].time := 900.0, [353].log_data[0].minminute := 30, [353].log_data[0].maxminute := 30, [353].log_data[0].valid := 1, [353].log_data[1].valid := 1, [353].log_data[2].valid := 1, [353].log_data[3].valid := 1, [353].log_data[4].valid := 1, [353].log_data[5].valid := 1, [353].log_data[6].valid := 1, [353].log_data[7].valid := 1, [353].log_data[8].valid := 1, [353].log_data[9].valid := 1, [353].log_data[10].valid := 1, [353].log_data[11].valid := 1, [353].log_data[12].valid := 1, [353].log_data[13].valid := 1, [353].log_data[14].valid := 1, [353].log_data[15].valid := 1, [353].log_data[16].valid := 1, [353].log_data[17].valid := 1, [353].log_data[18].valid := 1, [353].log_data[19].valid := 1, [353].time.Year := 2023, [353].time.Month := 1, [353].time.Day := 11, [353].time.Hour := 8, [353].time.Minute := 44, [353].time.Second := 59, [354].log_data[0].min := 1.0, [354].log_data[0].max := 1.0, [354].log_data[0].total := 900.0, [354].log_data[0].time := 900.0, [354].log_data[0].minminute := 45, [354].log_data[0].maxminute := 45, [354].log_data[0].valid := 1, [354].log_data[1].valid := 1, [354].log_data[2].valid := 1, [354].log_data[3].valid := 1, [354].log_data[4].valid := 1, [354].log_data[5].valid := 1, [354].log_data[6].valid := 1, [354].log_data[7].valid := 1, [354].log_data[8].valid := 1, [354].log_data[9].valid := 1, [354].log_data[10].valid := 1, [354].log_data[11].valid := 1, [354].log_data[12].valid := 1, [354].log_data[13].valid := 1, [354].log_data[14].valid := 1, [354].log_data[15].valid := 1, [354].log_data[16].valid := 1, [354].log_data[17].valid := 1, [354].log_data[18].valid := 1, [354].log_data[19].valid := 1, [354].time.Year := 2023, [354].time.Month := 1, [354].time.Day := 11,
        [354].time.Hour := 8, [354].time.Minute := 59, [354].time.Second := 59, [355].log_data[0].min := 1.0, [355].log_data[0].max := 1.0, [355].log_data[0].total := 900.0, [355].log_data[0].time := 900.0, [355].log_data[0].valid := 1, [355].log_data[1].valid := 1, [355].log_data[2].valid := 1, [355].log_data[3].valid := 1, [355].log_data[4].valid := 1, [355].log_data[5].valid := 1, [355].log_data[6].valid := 1, [355].log_data[7].valid := 1, [355].log_data[8].valid := 1, [355].log_data[9].valid := 1, [355].log_data[10].valid := 1, [355].log_data[11].valid := 1, [355].log_data[12].valid := 1, [355].log_data[13].valid := 1, [355].log_data[14].valid := 1, [355].log_data[15].valid := 1, [355].log_data[16].valid := 1, [355].log_data[17].valid := 1, [355].log_data[18].valid := 1, [355].log_data[19].valid := 1, [355].time.Year := 2023, [355].time.Month := 1, [355].time.Day := 11, [355].time.Hour := 9, [355].time.Minute := 14, [355].time.Second := 59, [356].log_data[0].min := 1.0, [356].log_data[0].max := 1.0, [356].log_data[0].total := 900.0, [356].log_data[0].time := 900.0, [356].log_data[0].minminute := 15, [356].log_data[0].maxminute := 15, [356].log_data[0].valid := 1, [356].log_data[1].valid := 1, [356].log_data[2].valid := 1, [356].log_data[3].valid := 1, [356].log_data[4].valid := 1, [356].log_data[5].valid := 1, [356].log_data[6].valid := 1, [356].log_data[7].valid := 1, [356].log_data[8].valid := 1, [356].log_data[9].valid := 1, [356].log_data[10].valid := 1, [356].log_data[11].valid := 1, [356].log_data[12].valid := 1, [356].log_data[13].valid := 1, [356].log_data[14].valid := 1, [356].log_data[15].valid := 1, [356].log_data[16].valid := 1, [356].log_data[17].valid := 1, [356].log_data[18].valid := 1, [356].log_data[19].valid := 1, [356].time.Year := 2023,
        [356].time.Month := 1, [356].time.Day := 11, [356].time.Hour := 9, [356].time.Minute := 29, [356].time.Second := 59, [357].log_data[0].min := 1.0, [357].log_data[0].max := 1.0, [357].log_data[0].total := 900.0, [357].log_data[0].time := 900.0, [357].log_data[0].minminute := 30, [357].log_data[0].maxminute := 30, [357].log_data[0].valid := 1, [357].log_data[1].valid := 1, [357].log_data[2].valid := 1, [357].log_data[3].valid := 1, [357].log_data[4].valid := 1, [357].log_data[5].valid := 1, [357].log_data[6].valid := 1, [357].log_data[7].valid := 1, [357].log_data[8].valid := 1, [357].log_data[9].valid := 1, [357].log_data[10].valid := 1, [357].log_data[11].valid := 1, [357].log_data[12].valid := 1, [357].log_data[13].valid := 1, [357].log_data[14].valid := 1, [357].log_data[15].valid := 1, [357].log_data[16].valid := 1, [357].log_data[17].valid := 1, [357].log_data[18].valid := 1, [357].log_data[19].valid := 1, [357].time.Year := 2023, [357].time.Month := 1, [357].time.Day := 11, [357].time.Hour := 9, [357].time.Minute := 44, [357].time.Second := 59, [358].log_data[0].min := 1.0, [358].log_data[0].max := 1.0, [358].log_data[0].total := 900.0, [358].log_data[0].time := 900.0, [358].log_data[0].minminute := 45, [358].log_data[0].maxminute := 45, [358].log_data[0].valid := 1, [358].log_data[1].valid := 1, [358].log_data[2].valid := 1, [358].log_data[3].valid := 1, [358].log_data[4].valid := 1, [358].log_data[5].valid := 1, [358].log_data[6].valid := 1, [358].log_data[7].valid := 1, [358].log_data[8].valid := 1, [358].log_data[9].valid := 1, [358].log_data[10].valid := 1, [358].log_data[11].valid := 1, [358].log_data[12].valid := 1, [358].log_data[13].valid := 1, [358].log_data[14].valid := 1, [358].log_data[15].valid := 1, [358].log_data[16].valid := 1,
        [358].log_data[17].valid := 1, [358].log_data[18].valid := 1, [358].log_data[19].valid := 1, [358].time.Year := 2023, [358].time.Month := 1, [358].time.Day := 11, [358].time.Hour := 9, [358].time.Minute := 59, [358].time.Second := 59, [359].log_data[0].min := 1.0, [359].log_data[0].max := 1.0, [359].log_data[0].total := 900.0, [359].log_data[0].time := 900.0, [359].log_data[0].valid := 1, [359].log_data[1].valid := 1, [359].log_data[2].valid := 1, [359].log_data[3].valid := 1, [359].log_data[4].valid := 1, [359].log_data[5].valid := 1, [359].log_data[6].valid := 1, [359].log_data[7].valid := 1, [359].log_data[8].valid := 1, [359].log_data[9].valid := 1, [359].log_data[10].valid := 1, [359].log_data[11].valid := 1, [359].log_data[12].valid := 1, [359].log_data[13].valid := 1, [359].log_data[14].valid := 1, [359].log_data[15].valid := 1, [359].log_data[16].valid := 1, [359].log_data[17].valid := 1, [359].log_data[18].valid := 1, [359].log_data[19].valid := 1, [359].time.Year := 2023, [359].time.Month := 1, [359].time.Day := 11, [359].time.Hour := 10, [359].time.Minute := 14, [359].time.Second := 59, [360].log_data[0].min := 1.0, [360].log_data[0].max := 1.0, [360].log_data[0].total := 900.0, [360].log_data[0].time := 900.0, [360].log_data[0].minminute := 15, [360].log_data[0].maxminute := 15, [360].log_data[0].valid := 1, [360].log_data[1].valid := 1, [360].log_data[2].valid := 1, [360].log_data[3].valid := 1, [360].log_data[4].valid := 1, [360].log_data[5].valid := 1, [360].log_data[6].valid := 1, [360].log_data[7].valid := 1, [360].log_data[8].valid := 1, [360].log_data[9].valid := 1, [360].log_data[10].valid := 1, [360].log_data[11].valid := 1, [360].log_data[12].valid := 1, [360].log_data[13].valid := 1, [360].log_data[14].valid := 1,
        [360].log_data[15].valid := 1, [360].log_data[16].valid := 1, [360].log_data[17].valid := 1, [360].log_data[18].valid := 1, [360].log_data[19].valid := 1, [360].time.Year := 2023, [360].time.Month := 1, [360].time.Day := 11, [360].time.Hour := 10, [360].time.Minute := 29, [360].time.Second := 59, [361].log_data[0].min := 1.0, [361].log_data[0].max := 1.0, [361].log_data[0].total := 900.0, [361].log_data[0].time := 900.0, [361].log_data[0].minminute := 30, [361].log_data[0].maxminute := 30, [361].log_data[0].valid := 1, [361].log_data[1].valid := 1, [361].log_data[2].valid := 1, [361].log_data[3].valid := 1, [361].log_data[4].valid := 1, [361].log_data[5].valid := 1, [361].log_data[6].valid := 1, [361].log_data[7].valid := 1, [361].log_data[8].valid := 1, [361].log_data[9].valid := 1, [361].log_data[10].valid := 1, [361].log_data[11].valid := 1, [361].log_data[12].valid := 1, [361].log_data[13].valid := 1, [361].log_data[14].valid := 1, [361].log_data[15].valid := 1, [361].log_data[16].valid := 1, [361].log_data[17].valid := 1, [361].log_data[18].valid := 1, [361].log_data[19].valid := 1, [361].time.Year := 2023, [361].time.Month := 1, [361].time.Day := 11, [361].time.Hour := 10, [361].time.Minute := 44, [361].time.Second := 59, [362].log_data[0].min := 1.0, [362].log_data[0].max := 1.0, [362].log_data[0].total := 900.0, [362].log_data[0].time := 900.0, [362].log_data[0].minminute := 45, [362].log_data[0].maxminute := 45, [362].log_data[0].valid := 1, [362].log_data[1].valid := 1, [362].log_data[2].valid := 1, [362].log_data[3].valid := 1, [362].log_data[4].valid := 1, [362].log_data[5].valid := 1, [362].log_data[6].valid := 1, [362].log_data[7].valid := 1, [362].log_data[8].valid := 1, [362].log_data[9].valid := 1, [362].log_data[10].valid := 1,
        [362].log_data[11].valid := 1, [362].log_data[12].valid := 1, [362].log_data[13].valid := 1, [362].log_data[14].valid := 1, [362].log_data[15].valid := 1, [362].log_data[16].valid := 1, [362].log_data[17].valid := 1, [362].log_data[18].valid := 1, [362].log_data[19].valid := 1, [362].time.Year := 2023, [362].time.Month := 1, [362].time.Day := 11, [362].time.Hour := 10, [362].time.Minute := 59, [362].time.Second := 59, [363].log_data[0].min := 1.0, [363].log_data[0].max := 1.0, [363].log_data[0].total := 900.0, [363].log_data[0].time := 900.0, [363].log_data[0].valid := 1, [363].log_data[1].valid := 1, [363].log_data[2].valid := 1, [363].log_data[3].valid := 1, [363].log_data[4].valid := 1, [363].log_data[5].valid := 1, [363].log_data[6].valid := 1, [363].log_data[7].valid := 1, [363].log_data[8].valid := 1, [363].log_data[9].valid := 1, [363].log_data[10].valid := 1, [363].log_data[11].valid := 1, [363].log_data[12].valid := 1, [363].log_data[13].valid := 1, [363].log_data[14].valid := 1, [363].log_data[15].valid := 1, [363].log_data[16].valid := 1, [363].log_data[17].valid := 1, [363].log_data[18].valid := 1, [363].log_data[19].valid := 1, [363].time.Year := 2023, [363].time.Month := 1, [363].time.Day := 11, [363].time.Hour := 11, [363].time.Minute := 14, [363].time.Second := 59, [364].log_data[0].min := 1.0, [364].log_data[0].max := 1.0, [364].log_data[0].total := 900.0, [364].log_data[0].time := 900.0, [364].log_data[0].minminute := 15, [364].log_data[0].maxminute := 15, [364].log_data[0].valid := 1, [364].log_data[1].valid := 1, [364].log_data[2].valid := 1, [364].log_data[3].valid := 1, [364].log_data[4].valid := 1, [364].log_data[5].valid := 1, [364].log_data[6].valid := 1, [364].log_data[7].valid := 1, [364].log_data[8].valid := 1,
        [364].log_data[9].valid := 1, [364].log_data[10].valid := 1, [364].log_data[11].valid := 1, [364].log_data[12].valid := 1, [364].log_data[13].valid := 1, [364].log_data[14].valid := 1, [364].log_data[15].valid := 1, [364].log_data[16].valid := 1, [364].log_data[17].valid := 1, [364].log_data[18].valid := 1, [364].log_data[19].valid := 1, [364].time.Year := 2023, [364].time.Month := 1, [364].time.Day := 11, [364].time.Hour := 11, [364].time.Minute := 29, [364].time.Second := 59, [365].log_data[0].min := 1.0, [365].log_data[0].max := 1.0, [365].log_data[0].total := 900.0, [365].log_data[0].time := 900.0, [365].log_data[0].minminute := 30, [365].log_data[0].maxminute := 30, [365].log_data[0].valid := 1, [365].log_data[1].valid := 1, [365].log_data[2].valid := 1, [365].log_data[3].valid := 1, [365].log_data[4].valid := 1, [365].log_data[5].valid := 1, [365].log_data[6].valid := 1, [365].log_data[7].valid := 1, [365].log_data[8].valid := 1, [365].log_data[9].valid := 1, [365].log_data[10].valid := 1, [365].log_data[11].valid := 1, [365].log_data[12].valid := 1, [365].log_data[13].valid := 1, [365].log_data[14].valid := 1, [365].log_data[15].valid := 1, [365].log_data[16].valid := 1, [365].log_data[17].valid := 1, [365].log_data[18].valid := 1, [365].log_data[19].valid := 1, [365].time.Year := 2023, [365].time.Month := 1, [365].time.Day := 11, [365].time.Hour := 11, [365].time.Minute := 44, [365].time.Second := 59, [366].log_data[0].min := 1.0, [366].log_data[0].max := 1.0, [366].log_data[0].total := 900.0, [366].log_data[0].time := 900.0, [366].log_data[0].minminute := 45, [366].log_data[0].maxminute := 45, [366].log_data[0].valid := 1, [366].log_data[1].valid := 1, [366].log_data[2].valid := 1, [366].log_data[3].valid := 1, [366].log_data[4].valid := 1,
        [366].log_data[5].valid := 1, [366].log_data[6].valid := 1, [366].log_data[7].valid := 1, [366].log_data[8].valid := 1, [366].log_data[9].valid := 1, [366].log_data[10].valid := 1, [366].log_data[11].valid := 1, [366].log_data[12].valid := 1, [366].log_data[13].valid := 1, [366].log_data[14].valid := 1, [366].log_data[15].valid := 1, [366].log_data[16].valid := 1, [366].log_data[17].valid := 1, [366].log_data[18].valid := 1, [366].log_data[19].valid := 1, [366].time.Year := 2023, [366].time.Month := 1, [366].time.Day := 11, [366].time.Hour := 11, [366].time.Minute := 59, [366].time.Second := 59, [367].log_data[0].min := 1.0, [367].log_data[0].max := 1.0, [367].log_data[0].total := 900.0, [367].log_data[0].time := 900.0, [367].log_data[0].valid := 1, [367].log_data[1].valid := 1, [367].log_data[2].valid := 1, [367].log_data[3].valid := 1, [367].log_data[4].valid := 1, [367].log_data[5].valid := 1, [367].log_data[6].valid := 1, [367].log_data[7].valid := 1, [367].log_data[8].valid := 1, [367].log_data[9].valid := 1, [367].log_data[10].valid := 1, [367].log_data[11].valid := 1, [367].log_data[12].valid := 1, [367].log_data[13].valid := 1, [367].log_data[14].valid := 1, [367].log_data[15].valid := 1, [367].log_data[16].valid := 1, [367].log_data[17].valid := 1, [367].log_data[18].valid := 1, [367].log_data[19].valid := 1, [367].time.Year := 2023, [367].time.Month := 1, [367].time.Day := 11, [367].time.Hour := 12, [367].time.Minute := 14, [367].time.Second := 59, [368].log_data[0].min := 1.0, [368].log_data[0].max := 1.0, [368].log_data[0].total := 900.0, [368].log_data[0].time := 900.0, [368].log_data[0].minminute := 15, [368].log_data[0].maxminute := 15, [368].log_data[0].valid := 1, [368].log_data[1].valid := 1, [368].log_data[2].valid := 1,
        [368].log_data[3].valid := 1, [368].log_data[4].valid := 1, [368].log_data[5].valid := 1, [368].log_data[6].valid := 1, [368].log_data[7].valid := 1, [368].log_data[8].valid := 1, [368].log_data[9].valid := 1, [368].log_data[10].valid := 1, [368].log_data[11].valid := 1, [368].log_data[12].valid := 1, [368].log_data[13].valid := 1, [368].log_data[14].valid := 1, [368].log_data[15].valid := 1, [368].log_data[16].valid := 1, [368].log_data[17].valid := 1, [368].log_data[18].valid := 1, [368].log_data[19].valid := 1, [368].time.Year := 2023, [368].time.Month := 1, [368].time.Day := 11, [368].time.Hour := 12, [368].time.Minute := 29, [368].time.Second := 59, [369].log_data[0].min := 1.0, [369].log_data[0].max := 1.0, [369].log_data[0].total := 900.0, [369].log_data[0].time := 900.0, [369].log_data[0].minminute := 30, [369].log_data[0].maxminute := 30, [369].log_data[0].valid := 1, [369].log_data[1].valid := 1, [369].log_data[2].valid := 1, [369].log_data[3].valid := 1, [369].log_data[4].valid := 1, [369].log_data[5].valid := 1, [369].log_data[6].valid := 1, [369].log_data[7].valid := 1, [369].log_data[8].valid := 1, [369].log_data[9].valid := 1, [369].log_data[10].valid := 1, [369].log_data[11].valid := 1, [369].log_data[12].valid := 1, [369].log_data[13].valid := 1, [369].log_data[14].valid := 1, [369].log_data[15].valid := 1, [369].log_data[16].valid := 1, [369].log_data[17].valid := 1, [369].log_data[18].valid := 1, [369].log_data[19].valid := 1, [369].time.Year := 2023, [369].time.Month := 1, [369].time.Day := 11, [369].time.Hour := 12, [369].time.Minute := 44, [369].time.Second := 59, [370].log_data[0].min := 1.0, [370].log_data[0].max := 1.0, [370].log_data[0].total := 900.0, [370].log_data[0].time := 900.0, [370].log_data[0].minminute := 45,
        [370].log_data[0].maxminute := 45, [370].log_data[0].valid := 1, [370].log_data[1].valid := 1, [370].log_data[2].valid := 1, [370].log_data[3].valid := 1, [370].log_data[4].valid := 1, [370].log_data[5].valid := 1, [370].log_data[6].valid := 1, [370].log_data[7].valid := 1, [370].log_data[8].valid := 1, [370].log_data[9].valid := 1, [370].log_data[10].valid := 1, [370].log_data[11].valid := 1, [370].log_data[12].valid := 1, [370].log_data[13].valid := 1, [370].log_data[14].valid := 1, [370].log_data[15].valid := 1, [370].log_data[16].valid := 1, [370].log_data[17].valid := 1, [370].log_data[18].valid := 1, [370].log_data[19].valid := 1, [370].time.Year := 2023, [370].time.Month := 1, [370].time.Day := 11, [370].time.Hour := 12, [370].time.Minute := 59, [370].time.Second := 59, [371].log_data[0].min := 1.0, [371].log_data[0].max := 1.0, [371].log_data[0].total := 900.0, [371].log_data[0].time := 900.0, [371].log_data[0].valid := 1, [371].log_data[1].valid := 1, [371].log_data[2].valid := 1, [371].log_data[3].valid := 1, [371].log_data[4].valid := 1, [371].log_data[5].valid := 1, [371].log_data[6].valid := 1, [371].log_data[7].valid := 1, [371].log_data[8].valid := 1, [371].log_data[9].valid := 1, [371].log_data[10].valid := 1, [371].log_data[11].valid := 1, [371].log_data[12].valid := 1, [371].log_data[13].valid := 1, [371].log_data[14].valid := 1, [371].log_data[15].valid := 1, [371].log_data[16].valid := 1, [371].log_data[17].valid := 1, [371].log_data[18].valid := 1, [371].log_data[19].valid := 1, [371].time.Year := 2023, [371].time.Month := 1, [371].time.Day := 11, [371].time.Hour := 13, [371].time.Minute := 14, [371].time.Second := 59, [372].log_data[0].min := 1.0, [372].log_data[0].max := 1.0, [372].log_data[0].total := 900.0,
        [372].log_data[0].time := 900.0, [372].log_data[0].minminute := 15, [372].log_data[0].maxminute := 15, [372].log_data[0].valid := 1, [372].log_data[1].valid := 1, [372].log_data[2].valid := 1, [372].log_data[3].valid := 1, [372].log_data[4].valid := 1, [372].log_data[5].valid := 1, [372].log_data[6].valid := 1, [372].log_data[7].valid := 1, [372].log_data[8].valid := 1, [372].log_data[9].valid := 1, [372].log_data[10].valid := 1, [372].log_data[11].valid := 1, [372].log_data[12].valid := 1, [372].log_data[13].valid := 1, [372].log_data[14].valid := 1, [372].log_data[15].valid := 1, [372].log_data[16].valid := 1, [372].log_data[17].valid := 1, [372].log_data[18].valid := 1, [372].log_data[19].valid := 1, [372].time.Year := 2023, [372].time.Month := 1, [372].time.Day := 11, [372].time.Hour := 13, [372].time.Minute := 29, [372].time.Second := 59, [373].log_data[0].min := 1.0, [373].log_data[0].max := 1.0, [373].log_data[0].total := 900.0, [373].log_data[0].time := 900.0, [373].log_data[0].minminute := 30, [373].log_data[0].maxminute := 30, [373].log_data[0].valid := 1, [373].log_data[1].valid := 1, [373].log_data[2].valid := 1, [373].log_data[3].valid := 1, [373].log_data[4].valid := 1, [373].log_data[5].valid := 1, [373].log_data[6].valid := 1, [373].log_data[7].valid := 1, [373].log_data[8].valid := 1, [373].log_data[9].valid := 1, [373].log_data[10].valid := 1, [373].log_data[11].valid := 1, [373].log_data[12].valid := 1, [373].log_data[13].valid := 1, [373].log_data[14].valid := 1, [373].log_data[15].valid := 1, [373].log_data[16].valid := 1, [373].log_data[17].valid := 1, [373].log_data[18].valid := 1, [373].log_data[19].valid := 1, [373].time.Year := 2023, [373].time.Month := 1, [373].time.Day := 11, [373].time.Hour := 13, [373].time.Minute := 44,
        [373].time.Second := 59, [374].log_data[0].min := 1.0, [374].log_data[0].max := 1.0, [374].log_data[0].total := 900.0, [374].log_data[0].time := 900.0, [374].log_data[0].minminute := 45, [374].log_data[0].maxminute := 45, [374].log_data[0].valid := 1, [374].log_data[1].valid := 1, [374].log_data[2].valid := 1, [374].log_data[3].valid := 1, [374].log_data[4].valid := 1, [374].log_data[5].valid := 1, [374].log_data[6].valid := 1, [374].log_data[7].valid := 1, [374].log_data[8].valid := 1, [374].log_data[9].valid := 1, [374].log_data[10].valid := 1, [374].log_data[11].valid := 1, [374].log_data[12].valid := 1, [374].log_data[13].valid := 1, [374].log_data[14].valid := 1, [374].log_data[15].valid := 1, [374].log_data[16].valid := 1, [374].log_data[17].valid := 1, [374].log_data[18].valid := 1, [374].log_data[19].valid := 1, [374].time.Year := 2023, [374].time.Month := 1, [374].time.Day := 11, [374].time.Hour := 13, [374].time.Minute := 59, [374].time.Second := 59, [375].log_data[0].min := 1.0, [375].log_data[0].max := 1.0, [375].log_data[0].total := 899.5, [375].log_data[0].time := 899.5, [375].log_data[0].valid := 1, [375].log_data[1].valid := 1, [375].log_data[2].valid := 1, [375].log_data[3].valid := 1, [375].log_data[4].valid := 1, [375].log_data[5].valid := 1, [375].log_data[6].valid := 1, [375].log_data[7].valid := 1, [375].log_data[8].valid := 1, [375].log_data[9].valid := 1, [375].log_data[10].valid := 1, [375].log_data[11].valid := 1, [375].log_data[12].valid := 1, [375].log_data[13].valid := 1, [375].log_data[14].valid := 1, [375].log_data[15].valid := 1, [375].log_data[16].valid := 1, [375].log_data[17].valid := 1, [375].log_data[18].valid := 1, [375].log_data[19].valid := 1, [375].time.Year := 2023, [375].time.Month := 1, [375].time.Day := 11,
        [375].time.Hour := 14, [375].time.Minute := 14, [375].time.Second := 59, [376].log_data[0].min := 1.0, [376].log_data[0].max := 1.0, [376].log_data[0].total := 900.0, [376].log_data[0].time := 900.0, [376].log_data[0].minminute := 15, [376].log_data[0].maxminute := 15, [376].log_data[0].valid := 1, [376].log_data[1].valid := 1, [376].log_data[2].valid := 1, [376].log_data[3].valid := 1, [376].log_data[4].valid := 1, [376].log_data[5].valid := 1, [376].log_data[6].valid := 1, [376].log_data[7].valid := 1, [376].log_data[8].valid := 1, [376].log_data[9].valid := 1, [376].log_data[10].valid := 1, [376].log_data[11].valid := 1, [376].log_data[12].valid := 1, [376].log_data[13].valid := 1, [376].log_data[14].valid := 1, [376].log_data[15].valid := 1, [376].log_data[16].valid := 1, [376].log_data[17].valid := 1, [376].log_data[18].valid := 1, [376].log_data[19].valid := 1, [376].time.Year := 2023, [376].time.Month := 1, [376].time.Day := 11, [376].time.Hour := 14, [376].time.Minute := 29, [376].time.Second := 59, [377].log_data[0].min := 1.0, [377].log_data[0].max := 1.0, [377].log_data[0].total := 900.0, [377].log_data[0].time := 900.0, [377].log_data[0].minminute := 30, [377].log_data[0].maxminute := 30, [377].log_data[0].valid := 1, [377].log_data[1].valid := 1, [377].log_data[2].valid := 1, [377].log_data[3].valid := 1, [377].log_data[4].valid := 1, [377].log_data[5].valid := 1, [377].log_data[6].valid := 1, [377].log_data[7].valid := 1, [377].log_data[8].valid := 1, [377].log_data[9].valid := 1, [377].log_data[10].valid := 1, [377].log_data[11].valid := 1, [377].log_data[12].valid := 1, [377].log_data[13].valid := 1, [377].log_data[14].valid := 1, [377].log_data[15].valid := 1, [377].log_data[16].valid := 1, [377].log_data[17].valid := 1, [377].log_data[18].valid := 1,
        [377].log_data[19].valid := 1, [377].time.Year := 2023, [377].time.Month := 1, [377].time.Day := 11, [377].time.Hour := 14, [377].time.Minute := 44, [377].time.Second := 59, [378].log_data[0].min := 1.0, [378].log_data[0].max := 1.0, [378].log_data[0].total := 900.0, [378].log_data[0].time := 900.0, [378].log_data[0].minminute := 45, [378].log_data[0].maxminute := 45, [378].log_data[0].valid := 1, [378].log_data[1].valid := 1, [378].log_data[2].valid := 1, [378].log_data[3].valid := 1, [378].log_data[4].valid := 1, [378].log_data[5].valid := 1, [378].log_data[6].valid := 1, [378].log_data[7].valid := 1, [378].log_data[8].valid := 1, [378].log_data[9].valid := 1, [378].log_data[10].valid := 1, [378].log_data[11].valid := 1, [378].log_data[12].valid := 1, [378].log_data[13].valid := 1, [378].log_data[14].valid := 1, [378].log_data[15].valid := 1, [378].log_data[16].valid := 1, [378].log_data[17].valid := 1, [378].log_data[18].valid := 1, [378].log_data[19].valid := 1, [378].time.Year := 2023, [378].time.Month := 1, [378].time.Day := 11, [378].time.Hour := 14, [378].time.Minute := 59, [378].time.Second := 59, [379].log_data[0].min := 1.0, [379].log_data[0].max := 1.0, [379].log_data[0].total := 900.0, [379].log_data[0].time := 900.0, [379].log_data[0].valid := 1, [379].log_data[1].valid := 1, [379].log_data[2].valid := 1, [379].log_data[3].valid := 1, [379].log_data[4].valid := 1, [379].log_data[5].valid := 1, [379].log_data[6].valid := 1, [379].log_data[7].valid := 1, [379].log_data[8].valid := 1, [379].log_data[9].valid := 1, [379].log_data[10].valid := 1, [379].log_data[11].valid := 1, [379].log_data[12].valid := 1, [379].log_data[13].valid := 1, [379].log_data[14].valid := 1, [379].log_data[15].valid := 1, [379].log_data[16].valid := 1,
        [379].log_data[17].valid := 1, [379].log_data[18].valid := 1, [379].log_data[19].valid := 1, [379].time.Year := 2023, [379].time.Month := 1, [379].time.Day := 11, [379].time.Hour := 15, [379].time.Minute := 14, [379].time.Second := 59, [380].log_data[0].min := 1.0, [380].log_data[0].max := 1.0, [380].log_data[0].total := 900.0, [380].log_data[0].time := 900.0, [380].log_data[0].minminute := 15, [380].log_data[0].maxminute := 15, [380].log_data[0].valid := 1, [380].log_data[1].valid := 1, [380].log_data[2].valid := 1, [380].log_data[3].valid := 1, [380].log_data[4].valid := 1, [380].log_data[5].valid := 1, [380].log_data[6].valid := 1, [380].log_data[7].valid := 1, [380].log_data[8].valid := 1, [380].log_data[9].valid := 1, [380].log_data[10].valid := 1, [380].log_data[11].valid := 1, [380].log_data[12].valid := 1, [380].log_data[13].valid := 1, [380].log_data[14].valid := 1, [380].log_data[15].valid := 1, [380].log_data[16].valid := 1, [380].log_data[17].valid := 1, [380].log_data[18].valid := 1, [380].log_data[19].valid := 1, [380].time.Year := 2023, [380].time.Month := 1, [380].time.Day := 11, [380].time.Hour := 15, [380].time.Minute := 29, [380].time.Second := 59, [381].log_data[0].min := 1.0, [381].log_data[0].max := 1.0, [381].log_data[0].total := 900.0, [381].log_data[0].time := 900.0, [381].log_data[0].minminute := 30, [381].log_data[0].maxminute := 30, [381].log_data[0].valid := 1, [381].log_data[1].valid := 1, [381].log_data[2].valid := 1, [381].log_data[3].valid := 1, [381].log_data[4].valid := 1, [381].log_data[5].valid := 1, [381].log_data[6].valid := 1, [381].log_data[7].valid := 1, [381].log_data[8].valid := 1, [381].log_data[9].valid := 1, [381].log_data[10].valid := 1, [381].log_data[11].valid := 1, [381].log_data[12].valid := 1,
        [381].log_data[13].valid := 1, [381].log_data[14].valid := 1, [381].log_data[15].valid := 1, [381].log_data[16].valid := 1, [381].log_data[17].valid := 1, [381].log_data[18].valid := 1, [381].log_data[19].valid := 1, [381].time.Year := 2023, [381].time.Month := 1, [381].time.Day := 11, [381].time.Hour := 15, [381].time.Minute := 44, [381].time.Second := 59, [382].log_data[0].min := 1.0, [382].log_data[0].max := 1.0, [382].log_data[0].total := 900.0, [382].log_data[0].time := 900.0, [382].log_data[0].minminute := 45, [382].log_data[0].maxminute := 45, [382].log_data[0].valid := 1, [382].log_data[1].valid := 1, [382].log_data[2].valid := 1, [382].log_data[3].valid := 1, [382].log_data[4].valid := 1, [382].log_data[5].valid := 1, [382].log_data[6].valid := 1, [382].log_data[7].valid := 1, [382].log_data[8].valid := 1, [382].log_data[9].valid := 1, [382].log_data[10].valid := 1, [382].log_data[11].valid := 1, [382].log_data[12].valid := 1, [382].log_data[13].valid := 1, [382].log_data[14].valid := 1, [382].log_data[15].valid := 1, [382].log_data[16].valid := 1, [382].log_data[17].valid := 1, [382].log_data[18].valid := 1, [382].log_data[19].valid := 1, [382].time.Year := 2023, [382].time.Month := 1, [382].time.Day := 11, [382].time.Hour := 15, [382].time.Minute := 59, [382].time.Second := 59, [383].log_data[0].min := 1.0, [383].log_data[0].max := 1.0, [383].log_data[0].total := 900.0, [383].log_data[0].time := 900.0, [383].log_data[0].valid := 1, [383].log_data[1].valid := 1, [383].log_data[2].valid := 1, [383].log_data[3].valid := 1, [383].log_data[4].valid := 1, [383].log_data[5].valid := 1, [383].log_data[6].valid := 1, [383].log_data[7].valid := 1, [383].log_data[8].valid := 1, [383].log_data[9].valid := 1, [383].log_data[10].valid := 1,
        [383].log_data[11].valid := 1, [383].log_data[12].valid := 1, [383].log_data[13].valid := 1, [383].log_data[14].valid := 1, [383].log_data[15].valid := 1, [383].log_data[16].valid := 1, [383].log_data[17].valid := 1, [383].log_data[18].valid := 1, [383].log_data[19].valid := 1, [383].time.Year := 2023, [383].time.Month := 1, [383].time.Day := 11, [383].time.Hour := 16, [383].time.Minute := 14, [383].time.Second := 59, [384].log_data[0].min := 1.0, [384].log_data[0].max := 1.0, [384].log_data[0].total := 900.0, [384].log_data[0].time := 900.0, [384].log_data[0].minminute := 15, [384].log_data[0].maxminute := 15, [384].log_data[0].valid := 1, [384].log_data[1].valid := 1, [384].log_data[2].valid := 1, [384].log_data[3].valid := 1, [384].log_data[4].valid := 1, [384].log_data[5].valid := 1, [384].log_data[6].valid := 1, [384].log_data[7].valid := 1, [384].log_data[8].valid := 1, [384].log_data[9].valid := 1, [384].log_data[10].valid := 1, [384].log_data[11].valid := 1, [384].log_data[12].valid := 1, [384].log_data[13].valid := 1, [384].log_data[14].valid := 1, [384].log_data[15].valid := 1, [384].log_data[16].valid := 1, [384].log_data[17].valid := 1, [384].log_data[18].valid := 1, [384].log_data[19].valid := 1, [384].time.Year := 2023, [384].time.Month := 1, [384].time.Day := 11, [384].time.Hour := 16, [384].time.Minute := 29, [384].time.Second := 59, [385].log_data[0].min := 1.0, [385].log_data[0].max := 1.0, [385].log_data[0].total := 900.0, [385].log_data[0].time := 900.0, [385].log_data[0].minminute := 30, [385].log_data[0].maxminute := 30, [385].log_data[0].valid := 1, [385].log_data[1].valid := 1, [385].log_data[2].valid := 1, [385].log_data[3].valid := 1, [385].log_data[4].valid := 1, [385].log_data[5].valid := 1, [385].log_data[6].valid := 1,
        [385].log_data[7].valid := 1, [385].log_data[8].valid := 1, [385].log_data[9].valid := 1, [385].log_data[10].valid := 1, [385].log_data[11].valid := 1, [385].log_data[12].valid := 1, [385].log_data[13].valid := 1, [385].log_data[14].valid := 1, [385].log_data[15].valid := 1, [385].log_data[16].valid := 1, [385].log_data[17].valid := 1, [385].log_data[18].valid := 1, [385].log_data[19].valid := 1, [385].time.Year := 2023, [385].time.Month := 1, [385].time.Day := 11, [385].time.Hour := 16, [385].time.Minute := 44, [385].time.Second := 59, [386].log_data[0].min := 1.0, [386].log_data[0].max := 1.0, [386].log_data[0].total := 900.0, [386].log_data[0].time := 900.0, [386].log_data[0].minminute := 45, [386].log_data[0].maxminute := 45, [386].log_data[0].valid := 1, [386].log_data[1].valid := 1, [386].log_data[2].valid := 1, [386].log_data[3].valid := 1, [386].log_data[4].valid := 1, [386].log_data[5].valid := 1, [386].log_data[6].valid := 1, [386].log_data[7].valid := 1, [386].log_data[8].valid := 1, [386].log_data[9].valid := 1, [386].log_data[10].valid := 1, [386].log_data[11].valid := 1, [386].log_data[12].valid := 1, [386].log_data[13].valid := 1, [386].log_data[14].valid := 1, [386].log_data[15].valid := 1, [386].log_data[16].valid := 1, [386].log_data[17].valid := 1, [386].log_data[18].valid := 1, [386].log_data[19].valid := 1, [386].time.Year := 2023, [386].time.Month := 1, [386].time.Day := 11, [386].time.Hour := 16, [386].time.Minute := 59, [386].time.Second := 59, [387].log_data[0].min := 1.0, [387].log_data[0].max := 1.0, [387].log_data[0].total := 900.0, [387].log_data[0].time := 900.0, [387].log_data[0].valid := 1, [387].log_data[1].valid := 1, [387].log_data[2].valid := 1, [387].log_data[3].valid := 1, [387].log_data[4].valid := 1,
        [387].log_data[5].valid := 1, [387].log_data[6].valid := 1, [387].log_data[7].valid := 1, [387].log_data[8].valid := 1, [387].log_data[9].valid := 1, [387].log_data[10].valid := 1, [387].log_data[11].valid := 1, [387].log_data[12].valid := 1, [387].log_data[13].valid := 1, [387].log_data[14].valid := 1, [387].log_data[15].valid := 1, [387].log_data[16].valid := 1, [387].log_data[17].valid := 1, [387].log_data[18].valid := 1, [387].log_data[19].valid := 1, [387].time.Year := 2023, [387].time.Month := 1, [387].time.Day := 11, [387].time.Hour := 17, [387].time.Minute := 14, [387].time.Second := 59, [388].log_data[0].min := 1.0, [388].log_data[0].max := 1.0, [388].log_data[0].total := 900.0, [388].log_data[0].time := 900.0, [388].log_data[0].minminute := 15, [388].log_data[0].maxminute := 15, [388].log_data[0].valid := 1, [388].log_data[1].valid := 1, [388].log_data[2].valid := 1, [388].log_data[3].valid := 1, [388].log_data[4].valid := 1, [388].log_data[5].valid := 1, [388].log_data[6].valid := 1, [388].log_data[7].valid := 1, [388].log_data[8].valid := 1, [388].log_data[9].valid := 1, [388].log_data[10].valid := 1, [388].log_data[11].valid := 1, [388].log_data[12].valid := 1, [388].log_data[13].valid := 1, [388].log_data[14].valid := 1, [388].log_data[15].valid := 1, [388].log_data[16].valid := 1, [388].log_data[17].valid := 1, [388].log_data[18].valid := 1, [388].log_data[19].valid := 1, [388].time.Year := 2023, [388].time.Month := 1, [388].time.Day := 11, [388].time.Hour := 17, [388].time.Minute := 29, [388].time.Second := 59, [389].log_data[0].min := 1.0, [389].log_data[0].max := 1.0, [389].log_data[0].total := 900.0, [389].log_data[0].time := 900.0, [389].log_data[0].minminute := 30, [389].log_data[0].maxminute := 30, [389].log_data[0].valid := 1,
        [389].log_data[1].valid := 1, [389].log_data[2].valid := 1, [389].log_data[3].valid := 1, [389].log_data[4].valid := 1, [389].log_data[5].valid := 1, [389].log_data[6].valid := 1, [389].log_data[7].valid := 1, [389].log_data[8].valid := 1, [389].log_data[9].valid := 1, [389].log_data[10].valid := 1, [389].log_data[11].valid := 1, [389].log_data[12].valid := 1, [389].log_data[13].valid := 1, [389].log_data[14].valid := 1, [389].log_data[15].valid := 1, [389].log_data[16].valid := 1, [389].log_data[17].valid := 1, [389].log_data[18].valid := 1, [389].log_data[19].valid := 1, [389].time.Year := 2023, [389].time.Month := 1, [389].time.Day := 11, [389].time.Hour := 17, [389].time.Minute := 44, [389].time.Second := 59, [390].log_data[0].min := 1.0, [390].log_data[0].max := 1.0, [390].log_data[0].total := 900.0, [390].log_data[0].time := 900.0, [390].log_data[0].minminute := 45, [390].log_data[0].maxminute := 45, [390].log_data[0].valid := 1, [390].log_data[1].valid := 1, [390].log_data[2].valid := 1, [390].log_data[3].valid := 1, [390].log_data[4].valid := 1, [390].log_data[5].valid := 1, [390].log_data[6].valid := 1, [390].log_data[7].valid := 1, [390].log_data[8].valid := 1, [390].log_data[9].valid := 1, [390].log_data[10].valid := 1, [390].log_data[11].valid := 1, [390].log_data[12].valid := 1, [390].log_data[13].valid := 1, [390].log_data[14].valid := 1, [390].log_data[15].valid := 1, [390].log_data[16].valid := 1, [390].log_data[17].valid := 1, [390].log_data[18].valid := 1, [390].log_data[19].valid := 1, [390].time.Year := 2023, [390].time.Month := 1, [390].time.Day := 11, [390].time.Hour := 17, [390].time.Minute := 59, [390].time.Second := 59, [391].log_data[0].min := 1.0, [391].log_data[0].max := 1.0, [391].log_data[0].total := 900.0,
        [391].log_data[0].time := 900.0, [391].log_data[0].valid := 1, [391].log_data[1].valid := 1, [391].log_data[2].valid := 1, [391].log_data[3].valid := 1, [391].log_data[4].valid := 1, [391].log_data[5].valid := 1, [391].log_data[6].valid := 1, [391].log_data[7].valid := 1, [391].log_data[8].valid := 1, [391].log_data[9].valid := 1, [391].log_data[10].valid := 1, [391].log_data[11].valid := 1, [391].log_data[12].valid := 1, [391].log_data[13].valid := 1, [391].log_data[14].valid := 1, [391].log_data[15].valid := 1, [391].log_data[16].valid := 1, [391].log_data[17].valid := 1, [391].log_data[18].valid := 1, [391].log_data[19].valid := 1, [391].time.Year := 2023, [391].time.Month := 1, [391].time.Day := 11, [391].time.Hour := 18, [391].time.Minute := 14, [391].time.Second := 59, [392].log_data[0].min := 1.0, [392].log_data[0].max := 1.0, [392].log_data[0].total := 900.0, [392].log_data[0].time := 900.0, [392].log_data[0].minminute := 15, [392].log_data[0].maxminute := 15, [392].log_data[0].valid := 1, [392].log_data[1].valid := 1, [392].log_data[2].valid := 1, [392].log_data[3].valid := 1, [392].log_data[4].valid := 1, [392].log_data[5].valid := 1, [392].log_data[6].valid := 1, [392].log_data[7].valid := 1, [392].log_data[8].valid := 1, [392].log_data[9].valid := 1, [392].log_data[10].valid := 1, [392].log_data[11].valid := 1, [392].log_data[12].valid := 1, [392].log_data[13].valid := 1, [392].log_data[14].valid := 1, [392].log_data[15].valid := 1, [392].log_data[16].valid := 1, [392].log_data[17].valid := 1, [392].log_data[18].valid := 1, [392].log_data[19].valid := 1, [392].time.Year := 2023, [392].time.Month := 1, [392].time.Day := 11, [392].time.Hour := 18, [392].time.Minute := 29, [392].time.Second := 59, [393].log_data[0].min := 1.0,
        [393].log_data[0].max := 1.0, [393].log_data[0].total := 900.0, [393].log_data[0].time := 900.0, [393].log_data[0].minminute := 30, [393].log_data[0].maxminute := 30, [393].log_data[0].valid := 1, [393].log_data[1].valid := 1, [393].log_data[2].valid := 1, [393].log_data[3].valid := 1, [393].log_data[4].valid := 1, [393].log_data[5].valid := 1, [393].log_data[6].valid := 1, [393].log_data[7].valid := 1, [393].log_data[8].valid := 1, [393].log_data[9].valid := 1, [393].log_data[10].valid := 1, [393].log_data[11].valid := 1, [393].log_data[12].valid := 1, [393].log_data[13].valid := 1, [393].log_data[14].valid := 1, [393].log_data[15].valid := 1, [393].log_data[16].valid := 1, [393].log_data[17].valid := 1, [393].log_data[18].valid := 1, [393].log_data[19].valid := 1, [393].time.Year := 2023, [393].time.Month := 1, [393].time.Day := 11, [393].time.Hour := 18, [393].time.Minute := 44, [393].time.Second := 59, [394].log_data[0].min := 1.0, [394].log_data[0].max := 1.0, [394].log_data[0].total := 900.0, [394].log_data[0].time := 900.0, [394].log_data[0].minminute := 45, [394].log_data[0].maxminute := 45, [394].log_data[0].valid := 1, [394].log_data[1].valid := 1, [394].log_data[2].valid := 1, [394].log_data[3].valid := 1, [394].log_data[4].valid := 1, [394].log_data[5].valid := 1, [394].log_data[6].valid := 1, [394].log_data[7].valid := 1, [394].log_data[8].valid := 1, [394].log_data[9].valid := 1, [394].log_data[10].valid := 1, [394].log_data[11].valid := 1, [394].log_data[12].valid := 1, [394].log_data[13].valid := 1, [394].log_data[14].valid := 1, [394].log_data[15].valid := 1, [394].log_data[16].valid := 1, [394].log_data[17].valid := 1, [394].log_data[18].valid := 1, [394].log_data[19].valid := 1, [394].time.Year := 2023, [394].time.Month := 1, [394].time.Day := 11,
        [394].time.Hour := 18, [394].time.Minute := 59, [394].time.Second := 59, [395].log_data[0].min := 1.0, [395].log_data[0].max := 1.0, [395].log_data[0].total := 900.0, [395].log_data[0].time := 900.0, [395].log_data[0].valid := 1, [395].log_data[1].valid := 1, [395].log_data[2].valid := 1, [395].log_data[3].valid := 1, [395].log_data[4].valid := 1, [395].log_data[5].valid := 1, [395].log_data[6].valid := 1, [395].log_data[7].valid := 1, [395].log_data[8].valid := 1, [395].log_data[9].valid := 1, [395].log_data[10].valid := 1, [395].log_data[11].valid := 1, [395].log_data[12].valid := 1, [395].log_data[13].valid := 1, [395].log_data[14].valid := 1, [395].log_data[15].valid := 1, [395].log_data[16].valid := 1, [395].log_data[17].valid := 1, [395].log_data[18].valid := 1, [395].log_data[19].valid := 1, [395].time.Year := 2023, [395].time.Month := 1, [395].time.Day := 11, [395].time.Hour := 19, [395].time.Minute := 14, [395].time.Second := 59, [396].log_data[0].min := 1.0, [396].log_data[0].max := 1.0, [396].log_data[0].total := 900.0, [396].log_data[0].time := 900.0, [396].log_data[0].minminute := 15, [396].log_data[0].maxminute := 15, [396].log_data[0].valid := 1, [396].log_data[1].valid := 1, [396].log_data[2].valid := 1, [396].log_data[3].valid := 1, [396].log_data[4].valid := 1, [396].log_data[5].valid := 1, [396].log_data[6].valid := 1, [396].log_data[7].valid := 1, [396].log_data[8].valid := 1, [396].log_data[9].valid := 1, [396].log_data[10].valid := 1, [396].log_data[11].valid := 1, [396].log_data[12].valid := 1, [396].log_data[13].valid := 1, [396].log_data[14].valid := 1, [396].log_data[15].valid := 1, [396].log_data[16].valid := 1, [396].log_data[17].valid := 1, [396].log_data[18].valid := 1, [396].log_data[19].valid := 1, [396].time.Year := 2023,
        [396].time.Month := 1, [396].time.Day := 11, [396].time.Hour := 19, [396].time.Minute := 29, [396].time.Second := 59, [397].log_data[0].min := 1.0, [397].log_data[0].max := 1.0, [397].log_data[0].total := 900.0, [397].log_data[0].time := 900.0, [397].log_data[0].minminute := 30, [397].log_data[0].maxminute := 30, [397].log_data[0].valid := 1, [397].log_data[1].valid := 1, [397].log_data[2].valid := 1, [397].log_data[3].valid := 1, [397].log_data[4].valid := 1, [397].log_data[5].valid := 1, [397].log_data[6].valid := 1, [397].log_data[7].valid := 1, [397].log_data[8].valid := 1, [397].log_data[9].valid := 1, [397].log_data[10].valid := 1, [397].log_data[11].valid := 1, [397].log_data[12].valid := 1, [397].log_data[13].valid := 1, [397].log_data[14].valid := 1, [397].log_data[15].valid := 1, [397].log_data[16].valid := 1, [397].log_data[17].valid := 1, [397].log_data[18].valid := 1, [397].log_data[19].valid := 1, [397].time.Year := 2023, [397].time.Month := 1, [397].time.Day := 11, [397].time.Hour := 19, [397].time.Minute := 44, [397].time.Second := 59, [398].log_data[0].min := 1.0, [398].log_data[0].max := 1.0, [398].log_data[0].total := 900.0, [398].log_data[0].time := 900.0, [398].log_data[0].minminute := 45, [398].log_data[0].maxminute := 45, [398].log_data[0].valid := 1, [398].log_data[1].valid := 1, [398].log_data[2].valid := 1, [398].log_data[3].valid := 1, [398].log_data[4].valid := 1, [398].log_data[5].valid := 1, [398].log_data[6].valid := 1, [398].log_data[7].valid := 1, [398].log_data[8].valid := 1, [398].log_data[9].valid := 1, [398].log_data[10].valid := 1, [398].log_data[11].valid := 1, [398].log_data[12].valid := 1, [398].log_data[13].valid := 1, [398].log_data[14].valid := 1, [398].log_data[15].valid := 1, [398].log_data[16].valid := 1,
        [398].log_data[17].valid := 1, [398].log_data[18].valid := 1, [398].log_data[19].valid := 1, [398].time.Year := 2023, [398].time.Month := 1, [398].time.Day := 11, [398].time.Hour := 19, [398].time.Minute := 59, [398].time.Second := 59, [399].log_data[0].min := 1.0, [399].log_data[0].max := 1.0, [399].log_data[0].total := 900.0, [399].log_data[0].time := 900.0, [399].log_data[0].valid := 1, [399].log_data[1].valid := 1, [399].log_data[2].valid := 1, [399].log_data[3].valid := 1, [399].log_data[4].valid := 1, [399].log_data[5].valid := 1, [399].log_data[6].valid := 1, [399].log_data[7].valid := 1, [399].log_data[8].valid := 1, [399].log_data[9].valid := 1, [399].log_data[10].valid := 1, [399].log_data[11].valid := 1, [399].log_data[12].valid := 1, [399].log_data[13].valid := 1, [399].log_data[14].valid := 1, [399].log_data[15].valid := 1, [399].log_data[16].valid := 1, [399].log_data[17].valid := 1, [399].log_data[18].valid := 1, [399].log_data[19].valid := 1, [399].time.Year := 2023, [399].time.Month := 1, [399].time.Day := 11, [399].time.Hour := 20, [399].time.Minute := 14, [399].time.Second := 59, [400].log_data[0].min := 1.0, [400].log_data[0].max := 1.0, [400].log_data[0].total := 900.0, [400].log_data[0].time := 900.0, [400].log_data[0].minminute := 15, [400].log_data[0].maxminute := 15, [400].log_data[0].valid := 1, [400].log_data[1].valid := 1, [400].log_data[2].valid := 1, [400].log_data[3].valid := 1, [400].log_data[4].valid := 1, [400].log_data[5].valid := 1, [400].log_data[6].valid := 1, [400].log_data[7].valid := 1, [400].log_data[8].valid := 1, [400].log_data[9].valid := 1, [400].log_data[10].valid := 1, [400].log_data[11].valid := 1, [400].log_data[12].valid := 1, [400].log_data[13].valid := 1, [400].log_data[14].valid := 1,
        [400].log_data[15].valid := 1, [400].log_data[16].valid := 1, [400].log_data[17].valid := 1, [400].log_data[18].valid := 1, [400].log_data[19].valid := 1, [400].time.Year := 2023, [400].time.Month := 1, [400].time.Day := 11, [400].time.Hour := 20, [400].time.Minute := 29, [400].time.Second := 59, [401].log_data[0].min := 1.0, [401].log_data[0].max := 1.0, [401].log_data[0].total := 900.0, [401].log_data[0].time := 900.0, [401].log_data[0].minminute := 30, [401].log_data[0].maxminute := 30, [401].log_data[0].valid := 1, [401].log_data[1].valid := 1, [401].log_data[2].valid := 1, [401].log_data[3].valid := 1, [401].log_data[4].valid := 1, [401].log_data[5].valid := 1, [401].log_data[6].valid := 1, [401].log_data[7].valid := 1, [401].log_data[8].valid := 1, [401].log_data[9].valid := 1, [401].log_data[10].valid := 1, [401].log_data[11].valid := 1, [401].log_data[12].valid := 1, [401].log_data[13].valid := 1, [401].log_data[14].valid := 1, [401].log_data[15].valid := 1, [401].log_data[16].valid := 1, [401].log_data[17].valid := 1, [401].log_data[18].valid := 1, [401].log_data[19].valid := 1, [401].time.Year := 2023, [401].time.Month := 1, [401].time.Day := 11, [401].time.Hour := 20, [401].time.Minute := 44, [401].time.Second := 59, [402].log_data[0].min := 1.0, [402].log_data[0].max := 1.0, [402].log_data[0].total := 900.0, [402].log_data[0].time := 900.0, [402].log_data[0].minminute := 45, [402].log_data[0].maxminute := 45, [402].log_data[0].valid := 1, [402].log_data[1].valid := 1, [402].log_data[2].valid := 1, [402].log_data[3].valid := 1, [402].log_data[4].valid := 1, [402].log_data[5].valid := 1, [402].log_data[6].valid := 1, [402].log_data[7].valid := 1, [402].log_data[8].valid := 1, [402].log_data[9].valid := 1, [402].log_data[10].valid := 1,
        [402].log_data[11].valid := 1, [402].log_data[12].valid := 1, [402].log_data[13].valid := 1, [402].log_data[14].valid := 1, [402].log_data[15].valid := 1, [402].log_data[16].valid := 1, [402].log_data[17].valid := 1, [402].log_data[18].valid := 1, [402].log_data[19].valid := 1, [402].time.Year := 2023, [402].time.Month := 1, [402].time.Day := 11, [402].time.Hour := 20, [402].time.Minute := 59, [402].time.Second := 59, [403].log_data[0].min := 1.0, [403].log_data[0].max := 1.0, [403].log_data[0].total := 900.0, [403].log_data[0].time := 900.0, [403].log_data[0].valid := 1, [403].log_data[1].valid := 1, [403].log_data[2].valid := 1, [403].log_data[3].valid := 1, [403].log_data[4].valid := 1, [403].log_data[5].valid := 1, [403].log_data[6].valid := 1, [403].log_data[7].valid := 1, [403].log_data[8].valid := 1, [403].log_data[9].valid := 1, [403].log_data[10].valid := 1, [403].log_data[11].valid := 1, [403].log_data[12].valid := 1, [403].log_data[13].valid := 1, [403].log_data[14].valid := 1, [403].log_data[15].valid := 1, [403].log_data[16].valid := 1, [403].log_data[17].valid := 1, [403].log_data[18].valid := 1, [403].log_data[19].valid := 1, [403].time.Year := 2023, [403].time.Month := 1, [403].time.Day := 11, [403].time.Hour := 21, [403].time.Minute := 14, [403].time.Second := 59, [404].log_data[0].min := 1.0, [404].log_data[0].max := 1.0, [404].log_data[0].total := 900.0, [404].log_data[0].time := 900.0, [404].log_data[0].minminute := 15, [404].log_data[0].maxminute := 15, [404].log_data[0].valid := 1, [404].log_data[1].valid := 1, [404].log_data[2].valid := 1, [404].log_data[3].valid := 1, [404].log_data[4].valid := 1, [404].log_data[5].valid := 1, [404].log_data[6].valid := 1, [404].log_data[7].valid := 1, [404].log_data[8].valid := 1,
        [404].log_data[9].valid := 1, [404].log_data[10].valid := 1, [404].log_data[11].valid := 1, [404].log_data[12].valid := 1, [404].log_data[13].valid := 1, [404].log_data[14].valid := 1, [404].log_data[15].valid := 1, [404].log_data[16].valid := 1, [404].log_data[17].valid := 1, [404].log_data[18].valid := 1, [404].log_data[19].valid := 1, [404].time.Year := 2023, [404].time.Month := 1, [404].time.Day := 11, [404].time.Hour := 21, [404].time.Minute := 29, [404].time.Second := 59, [405].log_data[0].min := 1.0, [405].log_data[0].max := 1.0, [405].log_data[0].total := 900.0, [405].log_data[0].time := 900.0, [405].log_data[0].minminute := 30, [405].log_data[0].maxminute := 30, [405].log_data[0].valid := 1, [405].log_data[1].valid := 1, [405].log_data[2].valid := 1, [405].log_data[3].valid := 1, [405].log_data[4].valid := 1, [405].log_data[5].valid := 1, [405].log_data[6].valid := 1, [405].log_data[7].valid := 1, [405].log_data[8].valid := 1, [405].log_data[9].valid := 1, [405].log_data[10].valid := 1, [405].log_data[11].valid := 1, [405].log_data[12].valid := 1, [405].log_data[13].valid := 1, [405].log_data[14].valid := 1, [405].log_data[15].valid := 1, [405].log_data[16].valid := 1, [405].log_data[17].valid := 1, [405].log_data[18].valid := 1, [405].log_data[19].valid := 1, [405].time.Year := 2023, [405].time.Month := 1, [405].time.Day := 11, [405].time.Hour := 21, [405].time.Minute := 44, [405].time.Second := 59, [406].log_data[0].min := 1.0, [406].log_data[0].max := 1.0, [406].log_data[0].total := 900.0, [406].log_data[0].time := 900.0, [406].log_data[0].minminute := 45, [406].log_data[0].maxminute := 45, [406].log_data[0].valid := 1, [406].log_data[1].valid := 1, [406].log_data[2].valid := 1, [406].log_data[3].valid := 1, [406].log_data[4].valid := 1,
        [406].log_data[5].valid := 1, [406].log_data[6].valid := 1, [406].log_data[7].valid := 1, [406].log_data[8].valid := 1, [406].log_data[9].valid := 1, [406].log_data[10].valid := 1, [406].log_data[11].valid := 1, [406].log_data[12].valid := 1, [406].log_data[13].valid := 1, [406].log_data[14].valid := 1, [406].log_data[15].valid := 1, [406].log_data[16].valid := 1, [406].log_data[17].valid := 1, [406].log_data[18].valid := 1, [406].log_data[19].valid := 1, [406].time.Year := 2023, [406].time.Month := 1, [406].time.Day := 11, [406].time.Hour := 21, [406].time.Minute := 59, [406].time.Second := 59, [407].log_data[0].min := 1.0, [407].log_data[0].max := 1.0, [407].log_data[0].total := 900.0, [407].log_data[0].time := 900.0, [407].log_data[0].valid := 1, [407].log_data[1].valid := 1, [407].log_data[2].valid := 1, [407].log_data[3].valid := 1, [407].log_data[4].valid := 1, [407].log_data[5].valid := 1, [407].log_data[6].valid := 1, [407].log_data[7].valid := 1, [407].log_data[8].valid := 1, [407].log_data[9].valid := 1, [407].log_data[10].valid := 1, [407].log_data[11].valid := 1, [407].log_data[12].valid := 1, [407].log_data[13].valid := 1, [407].log_data[14].valid := 1, [407].log_data[15].valid := 1, [407].log_data[16].valid := 1, [407].log_data[17].valid := 1, [407].log_data[18].valid := 1, [407].log_data[19].valid := 1, [407].time.Year := 2023, [407].time.Month := 1, [407].time.Day := 11, [407].time.Hour := 22, [407].time.Minute := 14, [407].time.Second := 59, [408].log_data[0].min := 1.0, [408].log_data[0].max := 1.0, [408].log_data[0].total := 900.0, [408].log_data[0].time := 900.0, [408].log_data[0].minminute := 15, [408].log_data[0].maxminute := 15, [408].log_data[0].valid := 1, [408].log_data[1].valid := 1, [408].log_data[2].valid := 1,
        [408].log_data[3].valid := 1, [408].log_data[4].valid := 1, [408].log_data[5].valid := 1, [408].log_data[6].valid := 1, [408].log_data[7].valid := 1, [408].log_data[8].valid := 1, [408].log_data[9].valid := 1, [408].log_data[10].valid := 1, [408].log_data[11].valid := 1, [408].log_data[12].valid := 1, [408].log_data[13].valid := 1, [408].log_data[14].valid := 1, [408].log_data[15].valid := 1, [408].log_data[16].valid := 1, [408].log_data[17].valid := 1, [408].log_data[18].valid := 1, [408].log_data[19].valid := 1, [408].time.Year := 2023, [408].time.Month := 1, [408].time.Day := 11, [408].time.Hour := 22, [408].time.Minute := 29, [408].time.Second := 59, [409].log_data[0].min := 1.0, [409].log_data[0].max := 1.0, [409].log_data[0].total := 900.0, [409].log_data[0].time := 900.0, [409].log_data[0].minminute := 30, [409].log_data[0].maxminute := 30, [409].log_data[0].valid := 1, [409].log_data[1].valid := 1, [409].log_data[2].valid := 1, [409].log_data[3].valid := 1, [409].log_data[4].valid := 1, [409].log_data[5].valid := 1, [409].log_data[6].valid := 1, [409].log_data[7].valid := 1, [409].log_data[8].valid := 1, [409].log_data[9].valid := 1, [409].log_data[10].valid := 1, [409].log_data[11].valid := 1, [409].log_data[12].valid := 1, [409].log_data[13].valid := 1, [409].log_data[14].valid := 1, [409].log_data[15].valid := 1, [409].log_data[16].valid := 1, [409].log_data[17].valid := 1, [409].log_data[18].valid := 1, [409].log_data[19].valid := 1, [409].time.Year := 2023, [409].time.Month := 1, [409].time.Day := 11, [409].time.Hour := 22, [409].time.Minute := 44, [409].time.Second := 59, [410].log_data[0].min := 1.0, [410].log_data[0].max := 1.0, [410].log_data[0].total := 900.0, [410].log_data[0].time := 900.0, [410].log_data[0].minminute := 45,
        [410].log_data[0].maxminute := 45, [410].log_data[0].valid := 1, [410].log_data[1].valid := 1, [410].log_data[2].valid := 1, [410].log_data[3].valid := 1, [410].log_data[4].valid := 1, [410].log_data[5].valid := 1, [410].log_data[6].valid := 1, [410].log_data[7].valid := 1, [410].log_data[8].valid := 1, [410].log_data[9].valid := 1, [410].log_data[10].valid := 1, [410].log_data[11].valid := 1, [410].log_data[12].valid := 1, [410].log_data[13].valid := 1, [410].log_data[14].valid := 1, [410].log_data[15].valid := 1, [410].log_data[16].valid := 1, [410].log_data[17].valid := 1, [410].log_data[18].valid := 1, [410].log_data[19].valid := 1, [410].time.Year := 2023, [410].time.Month := 1, [410].time.Day := 11, [410].time.Hour := 22, [410].time.Minute := 59, [410].time.Second := 59, [411].log_data[0].min := 1.0, [411].log_data[0].max := 1.0, [411].log_data[0].total := 900.0, [411].log_data[0].time := 900.0, [411].log_data[0].valid := 1, [411].log_data[1].valid := 1, [411].log_data[2].valid := 1, [411].log_data[3].valid := 1, [411].log_data[4].valid := 1, [411].log_data[5].valid := 1, [411].log_data[6].valid := 1, [411].log_data[7].valid := 1, [411].log_data[8].valid := 1, [411].log_data[9].valid := 1, [411].log_data[10].valid := 1, [411].log_data[11].valid := 1, [411].log_data[12].valid := 1, [411].log_data[13].valid := 1, [411].log_data[14].valid := 1, [411].log_data[15].valid := 1, [411].log_data[16].valid := 1, [411].log_data[17].valid := 1, [411].log_data[18].valid := 1, [411].log_data[19].valid := 1, [411].time.Year := 2023, [411].time.Month := 1, [411].time.Day := 11, [411].time.Hour := 23, [411].time.Minute := 14, [411].time.Second := 59, [412].log_data[0].min := 1.0, [412].log_data[0].max := 1.0, [412].log_data[0].total := 900.0,
        [412].log_data[0].time := 900.0, [412].log_data[0].minminute := 15, [412].log_data[0].maxminute := 15, [412].log_data[0].valid := 1, [412].log_data[1].valid := 1, [412].log_data[2].valid := 1, [412].log_data[3].valid := 1, [412].log_data[4].valid := 1, [412].log_data[5].valid := 1, [412].log_data[6].valid := 1, [412].log_data[7].valid := 1, [412].log_data[8].valid := 1, [412].log_data[9].valid := 1, [412].log_data[10].valid := 1, [412].log_data[11].valid := 1, [412].log_data[12].valid := 1, [412].log_data[13].valid := 1, [412].log_data[14].valid := 1, [412].log_data[15].valid := 1, [412].log_data[16].valid := 1, [412].log_data[17].valid := 1, [412].log_data[18].valid := 1, [412].log_data[19].valid := 1, [412].time.Year := 2023, [412].time.Month := 1, [412].time.Day := 11, [412].time.Hour := 23, [412].time.Minute := 29, [412].time.Second := 59, [413].log_data[0].min := 1.0, [413].log_data[0].max := 1.0, [413].log_data[0].total := 900.0, [413].log_data[0].time := 900.0, [413].log_data[0].minminute := 30, [413].log_data[0].maxminute := 30, [413].log_data[0].valid := 1, [413].log_data[1].valid := 1, [413].log_data[2].valid := 1, [413].log_data[3].valid := 1, [413].log_data[4].valid := 1, [413].log_data[5].valid := 1, [413].log_data[6].valid := 1, [413].log_data[7].valid := 1, [413].log_data[8].valid := 1, [413].log_data[9].valid := 1, [413].log_data[10].valid := 1, [413].log_data[11].valid := 1, [413].log_data[12].valid := 1, [413].log_data[13].valid := 1, [413].log_data[14].valid := 1, [413].log_data[15].valid := 1, [413].log_data[16].valid := 1, [413].log_data[17].valid := 1, [413].log_data[18].valid := 1, [413].log_data[19].valid := 1, [413].time.Year := 2023, [413].time.Month := 1, [413].time.Day := 11, [413].time.Hour := 23, [413].time.Minute := 44,
